KUKA KRL program: MyProgram_144().src

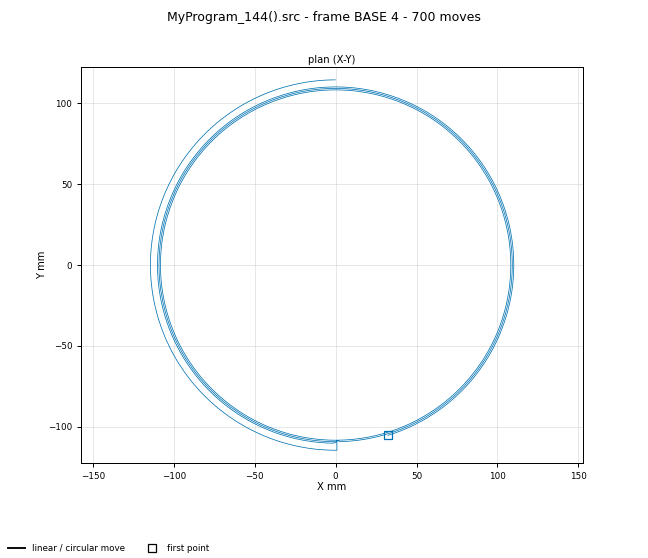
[picture p0: tool path of MyProgram_144().src in frame BASE 4, 700 of 700 moves have a stored position in this frame; points joined in program order, loops and branches not executed]
&ACCESS RVP
&REL 1
&PARAM TEMPLATE = C:\KRC\Roboter\Template\vorgabe
&PARAM EDITMASK = *
DEF MyProgram_144()
; ---- Setting reference (Base) ----
$BASE = BASE_DATA[4]

; --------------------------
; ---- Setting tool (TCP) ----
$TOOL = TOOL_DATA[3]
; --------------------------

$VEL.CP = VEL_APROX_PRINT
Startdeposition()
$VEL.CP = VEL_PRINT
LIN {X 32.3043,Y -105.2779,Z 114,A -76.1687,B 24.9494,C -1.6435,E1 25.049,E2 521.9318} C_DIS
LIN {X 36.8171,Y -103.7861,Z 114,A -73.6146,B 24.949,C -1.6502,E1 25.0557,E2 519.3669} C_DIS
LIN {X 40.1268,Y -102.5513,Z 114,A -71.7718,B 24.9488,C -1.6529,E1 25.0606,E2 517.5216} C_DIS
LIN {X 44.9405,Y -100.5354,Z 114,A -69.3366,B 24.9493,C -1.6447,E1 25.0667,E2 515.1116} C_DIS
LIN {X 48.2949,Y -98.9693,Z 114,A -67.5467,B 24.9495,C -1.6418,E1 25.0712,E2 513.3333} C_DIS
LIN {X 53.5849,Y -96.2059,Z 114,A -64.3362,B 24.9489,C -1.6518,E1 25.0792,E2 510.1083} C_DIS
LIN {X 56.8019,Y -94.3433,Z 114,A -62.2013,B 24.9481,C -1.6642,E1 25.0843,E2 507.9506} C_DIS
LIN {X 62.1001,Y -90.9432,Z 114,A -59.1184,B 24.9482,C -1.6622,E1 25.0915,E2 504.8827} C_DIS
LIN {X 65.0041,Y -88.8897,Z 114,A -57.5591,B 24.9488,C -1.6532,E1 25.095,E2 503.3502} C_DIS
LIN {X 67.0376,Y -87.3665,Z 114,A -55.8725,B 24.9476,C -1.6721,E1 25.0988,E2 501.6249} C_DIS
LIN {X 70.2691,Y -84.7891,Z 114,A -53.9266,B 24.9479,C -1.6678,E1 25.103,E2 499.6965} C_DIS
LIN {X 72.5045,Y -82.8856,Z 114,A -52.3507,B 24.9475,C -1.6735,E1 25.1063,E2 498.1135} C_DIS
LIN {X 75.3222,Y -80.3337,Z 114,A -50.387,B 24.9473,C -1.6775,E1 25.1104,E2 496.1481} C_DIS
LIN {X 77.8557,Y -77.8835,Z 114,A -48.461,B 24.9467,C -1.6861,E1 25.1142,E2 494.21} C_DIS
LIN {X 80.1666,Y -75.4999,Z 114,A -46.8371,B 24.9467,C -1.6859,E1 25.1174,E2 492.5937} C_DIS
LIN {X 82.7285,Y -72.6843,Z 114,A -44.8427,B 24.9464,C -1.6916,E1 25.1211,E2 490.5948} C_DIS
LIN {X 84.9909,Y -70.0262,Z 114,A -42.9743,B 24.9459,C -1.6987,E1 25.1244,E2 488.7181} C_DIS
LIN {X 87.034,Y -67.4692,Z 114,A -41.5863,B 24.9465,C -1.6892,E1 25.1268,E2 487.3591} C_DIS
LIN {X 88.7764,Y -65.1589,Z 114,A -39.9062,B 24.9458,C -1.7011,E1 25.1296,E2 485.6588} C_DIS
LIN {X 92.6081,Y -59.5874,Z 114,A -36.3603,B 24.9451,C -1.7122,E1 25.1352,E2 482.1042} C_DIS
LIN {X 95.3805,Y -55.0409,Z 114,A -33.6052,B 24.9446,C -1.7196,E1 25.1391,E2 479.346} C_DIS
LIN {X 97.1045,Y -51.9425,Z 114,A -30.8642,B 24.9416,C -1.7657,E1 25.1429,E2 476.5105} C_DIS
LIN {X 99.6138,Y -46.9497,Z 114,A -28.8531,B 24.9437,C -1.7337,E1 25.1452,E2 474.5857} C_DIS
LIN {X 100.9391,Y -44.025,Z 114,A -27.2776,B 24.9437,C -1.7345,E1 25.147,E2 473.0169} C_DIS
LIN {X 101.8876,Y -41.7839,Z 114,A -24.9103,B 24.94,C -1.7886,E1 25.1496,E2 470.535} C_DIS
LIN {X 104.1057,Y -35.9063,Z 114,A -21.5906,B 24.9392,C -1.8012,E1 25.1526,E2 467.2043} C_DIS
LIN {X 106.0459,Y -29.6867,Z 114,A -19.6143,B 24.9428,C -1.7475,E1 25.1541,E2 465.3661} C_DIS
LIN {X 106.6846,Y -27.3004,Z 114,A -17.8914,B 24.9412,C -1.7714,E1 25.1553,E2 463.5967} C_DIS
LIN {X 107.6606,Y -23.1559,Z 114,A -15.78,B 24.941,C -1.7738,E1 25.1566,E2 461.4918} C_DIS
LIN {X 108.3909,Y -19.4506,Z 114,A -13.9269,B 24.941,C -1.7751,E1 25.1575,E2 459.6465} C_DIS
LIN {X 109.0136,Y -15.5869,Z 114,A -11.905,B 24.9405,C -1.7811,E1 25.1584,E2 457.6225} C_DIS
LIN {X 109.4838,Y -11.8473,Z 114,A -10.1834,B 24.9408,C -1.7766,E1 25.1589,E2 455.9216} C_DIS
LIN {X 109.9148,Y -6.7857,Z 114,A -7.299,B 24.9395,C -1.7961,E1 25.1596,E2 453.0084} C_DIS
LIN {X 110.0683,Y -3.446,Z 114,A -5.6516,B 24.9395,C -1.7976,E1 25.1597,E2 451.3672} C_DIS
LIN {X 110.121,Y -0.6112,Z 114,A -3.8751,B 24.9382,C -1.816,E1 25.1597,E2 449.5578} C_DIS
LIN {X 110.0404,Y 4.2688,Z 114,A -1.5511,B 24.9382,C -1.8145,E1 25.1596,E2 447.2513} C_DIS
LIN {X 109.8312,Y 8.0234,Z 114,A 0.3876,B 24.9379,C -1.82,E1 25.1592,E2 445.3111} C_DIS
LIN {X 109.5211,Y 11.4902,Z 114,A 2.097,B 24.9379,C -1.8212,E1 25.1588,E2 443.609} C_DIS
LIN {X 109.109,Y 14.9152,Z 114,A 3.9492,B 24.9373,C -1.8295,E1 25.1581,E2 441.7481} C_DIS
LIN {X 108.6109,Y 18.1818,Z 114,A 5.5623,B 24.9373,C -1.8302,E1 25.1574,E2 440.1428} C_DIS
LIN {X 107.9638,Y 21.7008,Z 114,A 7.4442,B 24.9367,C -1.837,E1 25.1564,E2 438.256} C_DIS
LIN {X 107.3434,Y 24.5836,Z 114,A 8.962,B 24.9365,C -1.841,E1 25.1555,E2 436.7374} C_DIS
LIN {X 106.5404,Y 27.8614,Z 114,A 10.7334,B 24.936,C -1.8472,E1 25.1543,E2 434.9618} C_DIS
LIN {X 105.0229,Y 33.1235,Z 114,A 13.6108,B 24.9354,C -1.8571,E1 25.152,E2 432.0773} C_DIS
LIN {X 103.6854,Y 37.1036,Z 114,A 16.6543,B 24.9321,C -1.9024,E1 25.1491,E2 428.944} C_DIS
LIN {X 101.6602,Y 42.3358,Z 114,A 18.6311,B 24.9346,C -1.8684,E1 25.1471,E2 427.0584} C_DIS
LIN {X 100.4069,Y 45.2256,Z 114,A 20.2122,B 24.9344,C -1.8706,E1 25.1453,E2 425.4807} C_DIS
LIN {X 98.8908,Y 48.4539,Z 114,A 22.1571,B 24.9338,C -1.8798,E1 25.1429,E2 423.5245} C_DIS
LIN {X 97.2638,Y 51.6409,Z 114,A 24.2545,B 24.9326,C -1.8956,E1 25.1402,E2 421.4011} C_DIS
LIN {X 94.8756,Y 55.9067,Z 114,A 26.7935,B 24.9322,C -1.9022,E1 25.1366,E2 418.8594} C_DIS
LIN {X 92.3089,Y 60.0535,Z 114,A 29.0703,B 24.9325,C -1.8972,E1 25.1332,E2 416.6059} C_DIS
LIN {X 90.3472,Y 62.9628,Z 114,A 30.8213,B 24.9325,C -1.8986,E1 25.1305,E2 414.8602} C_DIS
LIN {X 88.2337,Y 65.8925,Z 114,A 32.6014,B 24.9325,C -1.8989,E1 25.1275,E2 413.088} C_DIS
LIN {X 84.6968,Y 70.3801,Z 114,A 35.6267,B 24.9317,C -1.9084,E1 25.1223,E2 410.0545} C_DIS
LIN {X 82.2831,Y 73.1882,Z 114,A 37.3292,B 24.9321,C -1.903,E1 25.1192,E2 408.3725} C_DIS
LIN {X 79.3562,Y 76.3512,Z 114,A 39.7796,B 24.9311,C -1.9171,E1 25.1145,E2 405.8994} C_DIS
LIN {X 76.8675,Y 78.8585,Z 114,A 41.7078,B 24.9305,C -1.9249,E1 25.1106,E2 403.9607} C_DIS
LIN {X 74.8797,Y 80.7482,Z 114,A 43.1989,B 24.9301,C -1.9307,E1 25.1075,E2 402.4622} C_DIS
LIN {X 71.615,Y 83.6557,Z 114,A 45.2986,B 24.9303,C -1.9276,E1 25.1032,E2 400.3781} C_DIS
LIN {X 68.7412,Y 86.0343,Z 114,A 47.3063,B 24.9299,C -1.9341,E1 25.0988,E2 398.3626} C_DIS
LIN {X 66.4134,Y 87.8424,Z 114,A 48.832,B 24.9297,C -1.9366,E1 25.0954,E2 396.8366} C_DIS
LIN {X 63.3023,Y 90.1112,Z 114,A 50.6227,B 24.9301,C -1.9308,E1 25.0914,E2 395.0658} C_DIS
LIN {X 60.4276,Y 92.0623,Z 114,A 52.8741,B 24.9285,C -1.953,E1 25.086,E2 392.7694} C_DIS
LIN {X 56.179,Y 94.7146,Z 114,A 55.3278,B 24.9287,C -1.9503,E1 25.0802,E2 390.3297} C_DIS
LIN {X 52.9765,Y 96.5437,Z 114,A 57.2821,B 24.9284,C -1.9545,E1 25.0754,E2 388.3712} C_DIS
LIN {X 48.8543,Y 98.6923,Z 114,A 59.4524,B 24.9289,C -1.947,E1 25.0701,E2 386.2246} C_DIS
LIN {X 45.5284,Y 100.2705,Z 114,A 61.4282,B 24.9286,C -1.9519,E1 25.0651,E2 384.2423} C_DIS
LIN {X 42.1119,Y 101.7542,Z 114,A 63.4155,B 24.9283,C -1.9561,E1 25.06,E2 382.2499} C_DIS
LIN {X 38.4349,Y 103.199,Z 114,A 66.0417,B 24.9263,C -1.9824,E1 25.053,E2 379.5669} C_DIS
LIN {X 34.2599,Y 104.6581,Z 114,A 67.6987,B 24.9282,C -1.9569,E1 25.0487,E2 377.9735} C_DIS
LIN {X 31.3328,Y 105.5707,Z 114,A 69.6145,B 24.9271,C -1.9717,E1 25.0435,E2 376.026} C_DIS
LIN {X 28.2462,Y 106.4392,Z 114,A 70.9701,B 24.928,C -1.9595,E1 25.0399,E2 374.7014} C_DIS
LIN {X 24.1237,Y 107.4495,Z 114,A 73.2559,B 24.9277,C -1.964,E1 25.0337,E2 372.4083} C_DIS
LIN {X 20.8233,Y 108.1356,Z 114,A 74.9128,B 24.9279,C -1.9607,E1 25.0292,E2 370.7611} C_DIS
LIN {X 16.9636,Y 108.8079,Z 114,A 76.9465,B 24.9279,C -1.9612,E1 25.0236,E2 368.7283} C_DIS
LIN {X 13.3331,Y 109.3134,Z 114,A 78.8773,B 24.9278,C -1.9626,E1 25.0182,E2 366.7957} C_DIS
LIN {X 9.9751,Y 109.6696,Z 114,A 80.606,B 24.9278,C -1.9617,E1 25.0134,E2 365.0704} C_DIS
LIN {X 6.296,Y 109.9423,Z 114,A 82.488,B 24.928,C -1.9601,E1 25.0082,E2 363.1928} C_DIS
LIN {X 2.8665,Y 110.0861,Z 114,A 84.3979,B 24.9276,C -1.9651,E1 25.0029,E2 361.2716} C_DIS
LIN {X -1.2189,Y 110.1168,Z 114,A 86.6393,B 24.9273,C -1.9694,E1 24.9966,E2 359.0199} C_DIS
LIN {X -5.4605,Y 109.9885,Z 114,A 88.6972,B 24.9278,C -1.9625,E1 24.9909,E2 356.978} C_DIS
LIN {X -8.5049,Y 109.7936,Z 114,A 90.2731,B 24.9278,C -1.9614,E1 24.9865,E2 355.4041} C_DIS
LIN {X -12.1976,Y 109.4464,Z 114,A 92.2543,B 24.9278,C -1.9625,E1 24.981,E2 353.4193} C_DIS
LIN {X -15.6118,Y 109.0101,Z 114,A 93.9501,B 24.9282,C -1.9575,E1 24.9763,E2 351.734} C_DIS
LIN {X -19.42,Y 108.3964,Z 114,A 95.7853,B 24.9288,C -1.9491,E1 24.9713,E2 349.9171} C_DIS
LIN {X -21.8574,Y 107.9317,Z 114,A 97.339,B 24.9281,C -1.9586,E1 24.967,E2 348.3389} C_DIS
LIN {X -26.1701,Y 106.9675,Z 114,A 100.5463,B 24.9255,C -1.9934,E1 24.9581,E2 345.0444} C_DIS
LIN {X -31.8564,Y 105.4153,Z 114,A 102.4384,B 24.9293,C -1.9424,E1 24.9533,E2 343.2705} C_DIS
LIN {X -37.6236,Y 103.4958,Z 114,A 105.8017,B 24.929,C -1.9465,E1 24.9444,E2 339.8911} C_DIS
LIN {X -40.94,Y 102.2311,Z 114,A 107.8444,B 24.9286,C -1.9518,E1 24.939,E2 337.8314} C_DIS
LIN {X -45.7047,Y 100.1911,Z 114,A 110.3935,B 24.9293,C -1.9419,E1 24.9325,E2 335.2997} C_DIS
LIN {X -48.9868,Y 98.6266,Z 114,A 112.713,B 24.9283,C -1.9559,E1 24.9266,E2 332.9408} C_DIS
LIN {X -52.1981,Y 96.9659,Z 114,A 114.2258,B 24.9296,C -1.9381,E1 24.923,E2 331.4662} C_DIS
LIN {X -55.7337,Y 94.9778,Z 114,A 116.2797,B 24.93,C -1.9321,E1 24.918,E2 329.4206} C_DIS
LIN {X -58.5565,Y 93.2637,Z 114,A 118.0509,B 24.93,C -1.931,E1 24.9138,E2 327.6464} C_DIS
LIN {X -61.885,Y 91.0888,Z 114,A 120.5693,B 24.9291,C -1.9446,E1 24.9079,E2 325.0872} C_DIS
LIN {X -64.9693,Y 88.9152,Z 114,A 122.0298,B 24.9308,C -1.9208,E1 24.9047,E2 323.6783} C_DIS
LIN {X -67.8244,Y 86.7588,Z 114,A 124.2205,B 24.9302,C -1.9297,E1 24.8998,E2 321.4584} C_DIS
LIN {X -71.8749,Y 83.4329,Z 114,A 127.1043,B 24.9302,C -1.9297,E1 24.8936,E2 318.5633} C_DIS
LIN {X -74.7712,Y 80.8477,Z 114,A 129.0145,B 24.9308,C -1.9207,E1 24.8897,E2 316.6669} C_DIS
LIN {X -78.7649,Y 76.9634,Z 114,A 131.8119,B 24.9316,C -1.9097,E1 24.8842,E2 313.8839} C_DIS
LIN {X -82.4622,Y 72.9882,Z 114,A 134.3424,B 24.933,C -1.8911,E1 24.8795,E2 311.3865} C_DIS
LIN {X -86.3423,Y 68.3515,Z 114,A 137.5194,B 24.9335,C -1.8841,E1 24.8739,E2 308.2116} C_DIS
LIN {X -89.6491,Y 63.9527,Z 114,A 140.4476,B 24.9338,C -1.8787,E1 24.869,E2 305.282} C_DIS
LIN {X -91.6855,Y 60.9991,Z 114,A 142.1773,B 24.9346,C -1.8683,E1 24.8663,E2 303.5687} C_DIS
LIN {X -94.787,Y 56.0565,Z 114,A 145.3711,B 24.9348,C -1.8656,E1 24.8616,E2 300.365} C_DIS
LIN {X -96.5285,Y 53.0045,Z 114,A 147.3129,B 24.9348,C -1.8646,E1 24.859,E2 298.4155} C_DIS
LIN {X -98.0542,Y 50.1226,Z 114,A 148.976,B 24.9353,C -1.8583,E1 24.8568,E2 296.7584} C_DIS
LIN {X -99.6777,Y 46.8124,Z 114,A 150.7436,B 24.9361,C -1.8467,E1 24.8547,E2 295.0088} C_DIS
LIN {X -101.664,Y 42.325,Z 114,A 153.4901,B 24.9361,C -1.8463,E1 24.8516,E2 292.2482} C_DIS
LIN {X -103.2769,Y 38.2238,Z 114,A 155.8023,B 24.9365,C -1.8399,E1 24.8493,E2 289.9382} C_DIS
LIN {X -104.3896,Y 35.0675,Z 114,A 157.4971,B 24.937,C -1.8327,E1 24.8478,E2 288.251} C_DIS
LIN {X -105.7838,Y 30.6115,Z 114,A 159.8834,B 24.9377,C -1.8233,E1 24.8459,E2 285.8732} C_DIS
LIN {X -107.2194,Y 25.1202,Z 114,A 162.9721,B 24.938,C -1.8191,E1 24.8437,E2 282.7767} C_DIS
LIN {X -107.9408,Y 21.8131,Z 114,A 164.6153,B 24.9387,C -1.8089,E1 24.8428,E2 281.148} C_DIS
LIN {X -108.5292,Y 18.6704,Z 114,A 166.8727,B 24.9375,C -1.8263,E1 24.8417,E2 278.8358} C_DIS
LIN {X -109.0902,Y 15.0478,Z 114,A 168.3564,B 24.939,C -1.8038,E1 24.8411,E2 277.3968} C_DIS
LIN {X -109.5684,Y 11.0388,Z 114,A 171.0753,B 24.9379,C -1.8208,E1 24.8403,E2 274.6212} C_DIS
LIN {X -109.9232,Y 6.6412,Z 114,A 172.611,B 24.9403,C -1.7842,E1 24.84,E2 273.1636} C_DIS
LIN {X -110.1166,Y 1.2654,Z 114,A 175.6442,B 24.9403,C -1.784,E1 24.8398,E2 270.1125} C_DIS
LIN {X -110.1145,Y -1.4343,Z 114,A 177.5079,B 24.9395,C -1.797,E1 24.8398,E2 268.2065} C_DIS
LIN {X -109.9939,Y -5.3508,Z 114,A 179.6017,B 24.9398,C -1.7926,E1 24.8402,E2 266.1107} C_DIS
LIN {X -109.7194,Y -9.4331,Z 114,A -178.7292,B 24.9414,C -1.768,E1 24.8405,E2 264.4901} C_DIS
LIN {X -109.4356,Y -12.2892,Z 114,A -176.8146,B 24.9407,C -1.7795,E1 24.8411,E2 262.5368} C_DIS
LIN {X -108.9413,Y -16.0959,Z 114,A -174.526,B 24.9403,C -1.7844,E1 24.8421,E2 260.2228} C_DIS
LIN {X -108.1152,Y -20.9288,Z 114,A -172.7875,B 24.9429,C -1.745,E1 24.8429,E2 258.5679} C_DIS
LIN {X -107.4211,Y -24.2447,Z 114,A -170.4746,B 24.9419,C -1.7607,E1 24.8444,E2 256.204} C_DIS
LIN {X -106.5292,Y -27.9049,Z 114,A -169.0976,B 24.9438,C -1.7322,E1 24.8453,E2 254.887} C_DIS
LIN {X -105.353,Y -32.0623,Z 114,A -166.6816,B 24.9438,C -1.7318,E1 24.8472,E2 252.458} C_DIS
LIN {X -104.4295,Y -34.9492,Z 114,A -165.129,B 24.9442,C -1.7261,E1 24.8485,E2 250.9101} C_DIS
LIN {X -103.2142,Y -38.3948,Z 114,A -163.1248,B 24.9442,C -1.7244,E1 24.8505,E2 248.8986} C_DIS
LIN {X -101.9882,Y -41.5368,Z 114,A -161.506,B 24.9449,C -1.714,E1 24.8521,E2 247.2955} C_DIS
LIN {X -100.8823,Y -44.1553,Z 114,A -159.764,B 24.9446,C -1.7199,E1 24.8541,E2 245.5297} C_DIS
LIN {X -98.8822,Y -48.4712,Z 114,A -157.6551,B 24.9459,C -1.6987,E1 24.8566,E2 243.4599} C_DIS
LIN {X -96.0493,Y -53.8654,Z 114,A -154.3168,B 24.9461,C -1.6964,E1 24.861,E2 240.1093} C_DIS
LIN {X -94.2141,Y -57.0145,Z 114,A -152.4164,B 24.9464,C -1.6915,E1 24.8637,E2 238.2109} C_DIS
LIN {X -92.8152,Y -59.2648,Z 114,A -150.2729,B 24.9447,C -1.718,E1 24.867,E2 235.9935} C_DIS
LIN {X -90.1561,Y -63.2377,Z 114,A -148.6355,B 24.9472,C -1.6782,E1 24.8695,E2 234.4428} C_DIS
LIN {X -86.1979,Y -68.5342,Z 114,A -144.9571,B 24.9472,C -1.679,E1 24.8757,E2 230.7448} C_DIS
LIN {X -83.7989,Y -71.4469,Z 114,A -143.0621,B 24.9476,C -1.6717,E1 24.8791,E2 228.8584} C_DIS
LIN {X -81.2882,Y -74.2912,Z 114,A -141.0843,B 24.9479,C -1.6674,E1 24.8828,E2 226.8821} C_DIS
LIN {X -78.8459,Y -76.8806,Z 114,A -139.1261,B 24.9479,C -1.6676,E1 24.8866,E2 224.9151} C_DIS
LIN {X -76.2978,Y -79.4077,Z 114,A -137.3686,B 24.9484,C -1.6593,E1 24.8901,E2 223.1699} C_DIS
LIN {X -73.573,Y -81.9387,Z 114,A -135.4544,B 24.9487,C -1.6546,E1 24.894,E2 221.2592} C_DIS
LIN {X -71.2807,Y -83.9404,Z 114,A -133.8601,B 24.9489,C -1.6519,E1 24.8974,E2 219.665} C_DIS
LIN {X -68.24,Y -86.4304,Z 114,A -131.7141,B 24.9489,C -1.6522,E1 24.9021,E2 217.5105} C_DIS
LIN {X -64.5235,Y -89.2394,Z 114,A -128.7329,B 24.9477,C -1.6704,E1 24.9089,E2 214.4754} C_DIS
LIN {X -61.0407,Y -91.658,Z 114,A -127.0719,B 24.9493,C -1.6447,E1 24.9126,E2 212.8698} C_DIS
LIN {X -58.565,Y -93.2584,Z 114,A -125.4735,B 24.9493,C -1.645,E1 24.9164,E2 211.2657} C_DIS
LIN {X -54.9688,Y -95.422,Z 114,A -123.3359,B 24.9496,C -1.64,E1 24.9215,E2 209.1337} C_DIS
LIN {X -51.4578,Y -97.3603,Z 114,A -121.2817,B 24.9499,C -1.6358,E1 24.9266,E2 207.0834} C_DIS
LIN {X -48.1628,Y -99.0329,Z 114,A -119.3115,B 24.9499,C -1.6354,E1 24.9315,E2 205.1092} C_DIS
LIN {X -44.9881,Y -100.5139,Z 114,A -117.4397,B 24.9499,C -1.6354,E1 24.9363,E2 203.2328} C_DIS
LIN {X -41.4514,Y -102.023,Z 114,A -114.8671,B 24.9486,C -1.6568,E1 24.9431,E2 200.6034} C_DIS
LIN {X -37.1934,Y -103.6527,Z 114,A -113.0418,B 24.9501,C -1.6321,E1 24.9477,E2 198.8332} C_DIS
LIN {X -34.4931,Y -104.5826,Z 114,A -111.2971,B 24.9495,C -1.6416,E1 24.9524,E2 197.0627} C_DIS
LIN {X -29.5647,Y -106.0805,Z 114,A -108.913,B 24.9504,C -1.6275,E1 24.9587,E2 194.7082} C_DIS
LIN {X -25.9792,Y -107.014,Z 114,A -107.0587,B 24.9506,C -1.6234,E1 24.9637,E2 192.8611} C_DIS
LIN {X -22.304,Y -107.84,Z 114,A -105.1248,B 24.9507,C -1.6214,E1 24.969,E2 190.9295} C_DIS
LIN {X -19.2869,Y -108.4203,Z 114,A -103.4094,B 24.9505,C -1.6257,E1 24.9737,E2 189.2021} C_DIS
LIN {X -15.5621,Y -109.0171,Z 114,A -101.7026,B 24.9512,C -1.6145,E1 24.9784,E2 187.5204} C_DIS
LIN {X -12.9079,Y -109.3632,Z 114,A -100.0154,B 24.9504,C -1.6266,E1 24.9831,E2 185.8033} C_DIS
LIN {X -8.8652,Y -109.7648,Z 114,A -98.0132,B 24.9507,C -1.6218,E1 24.9887,E2 183.8116} C_DIS
LIN {X -5.174,Y -110.0015,Z 114,A -95.9134,B 24.9503,C -1.6292,E1 24.9946,E2 181.6934} C_DIS
LIN {X -1.4311,Y -110.1144,Z 114,A -93.8231,B 24.9499,C -1.6356,E1 25.0005,E2 179.588} C_DIS
LIN {X -1.4311,Y -110.1144,Z 114,A -93.8231,B 24.9499,C -1.6356,E1 25.0005,E2 179.588} C_DIS
Enddeposition()
LIN {X 0.7939,Y -109.1989,Z 114,A -93.7268,B 24.9516,C -1.6074,E1 25.0005,E2 179.5585} C_DIS
Startdeposition()
$VEL.CP = VEL_PRINT
LIN {X -2.3355,Y -109.1788,Z 114,A -95.4072,B 24.9517,C -1.6054,E1 24.9958,E2 181.2435} C_DIS
LIN {X -5.5453,Y -109.0635,Z 114,A -97.1733,B 24.9519,C -1.6019,E1 24.9909,E2 183.0183} C_DIS
LIN {X -8.9577,Y -108.8356,Z 114,A -99.0359,B 24.9521,C -1.5992,E1 24.9857,E2 184.8882} C_DIS
LIN {X -13.2398,Y -108.3991,Z 114,A -101.142,B 24.9517,C -1.6057,E1 24.9799,E2 186.9802} C_DIS
LIN {X -16.5899,Y -107.9358,Z 114,A -102.9711,B 24.9517,C -1.6039,E1 24.9748,E2 188.8151} C_DIS
LIN {X -19.8828,Y -107.3795,Z 114,A -104.7313,B 24.9517,C -1.6041,E1 24.97,E2 190.5765} C_DIS
LIN {X -23.1749,Y -106.716,Z 114,A -106.4887,B 24.9517,C -1.6051,E1 24.9652,E2 192.3337} C_DIS
LIN {X -26.8944,Y -105.8402,Z 114,A -108.9002,B 24.9526,C -1.5899,E1 24.9585,E2 194.7847} C_DIS
LIN {X -30.1456,Y -104.9607,Z 114,A -110.0448,B 24.9511,C -1.616,E1 24.9556,E2 195.869} C_DIS
LIN {X -32.8817,Y -104.1368,Z 114,A -111.6886,B 24.9514,C -1.6113,E1 24.9512,E2 197.5269} C_DIS
LIN {X -35.7855,Y -103.1742,Z 114,A -113.4553,B 24.9517,C -1.6061,E1 24.9465,E2 199.3091} C_DIS
LIN {X -39.9101,Y -101.6491,Z 114,A -115.7497,B 24.9515,C -1.6088,E1 24.9405,E2 201.602} C_DIS
LIN {X -43.5494,Y -100.144,Z 114,A -117.8093,B 24.9514,C -1.6112,E1 24.9352,E2 203.6606} C_DIS
LIN {X -46.9166,Y -98.6122,Z 114,A -119.7309,B 24.9512,C -1.6143,E1 24.9303,E2 205.5798} C_DIS
LIN {X -49.9986,Y -97.0856,Z 114,A -121.5805,B 24.9512,C -1.6148,E1 24.9257,E2 207.4332} C_DIS
LIN {X -53.3124,Y -95.3056,Z 114,A -123.4281,B 24.9507,C -1.6224,E1 24.9212,E2 209.2678} C_DIS
LIN {X -56.1484,Y -93.6652,Z 114,A -125.305,B 24.9509,C -1.6186,E1 24.9166,E2 211.1594} C_DIS
LIN {X -58.983,Y -91.9041,Z 114,A -126.9357,B 24.9505,C -1.6261,E1 24.9128,E2 212.7775} C_DIS
LIN {X -65.0029,Y -87.7517,Z 114,A -130.7119,B 24.9499,C -1.6348,E1 24.9042,E2 216.5458} C_DIS
LIN {X -69.3844,Y -84.3295,Z 114,A -133.6115,B 24.9495,C -1.6408,E1 24.8979,E2 219.4419} C_DIS
LIN {X -71.6363,Y -82.4237,Z 114,A -135.3245,B 24.9498,C -1.6374,E1 24.8942,E2 221.1697} C_DIS
LIN {X -74.2905,Y -80.0417,Z 114,A -137.2983,B 24.9498,C -1.6372,E1 24.8901,E2 223.1519} C_DIS
LIN {X -76.8751,Y -77.5604,Z 114,A -139.0531,B 24.9492,C -1.646,E1 24.8866,E2 224.8931} C_DIS
LIN {X -79.4418,Y -74.9292,Z 114,A -141.0039,B 24.949,C -1.6494,E1 24.8828,E2 226.8444} C_DIS
LIN {X -81.8339,Y -72.3116,Z 114,A -142.9819,B 24.949,C -1.649,E1 24.8791,E2 228.8319} C_DIS
LIN {X -84.098,Y -69.6629,Z 114,A -144.6807,B 24.9485,C -1.6583,E1 24.8761,E2 230.5165} C_DIS
LIN {X -86.9831,Y -66.0273,Z 114,A -147.0336,B 24.9479,C -1.6673,E1 24.8721,E2 232.8591} C_DIS
LIN {X -89.2747,Y -62.8953,Z 114,A -149.3147,B 24.9482,C -1.663,E1 24.8683,E2 235.1614} C_DIS
LIN {X -91.7931,Y -59.1559,Z 114,A -151.292,B 24.9469,C -1.6839,E1 24.8653,E2 237.0988} C_DIS
LIN {X -93.1935,Y -56.9244,Z 114,A -153.0288,B 24.9475,C -1.6741,E1 24.8627,E2 238.868} C_DIS
LIN {X -95.124,Y -53.6376,Z 114,A -155.7701,B 24.9489,C -1.6517,E1 24.8588,E2 241.6771} C_DIS
LIN {X -97.4136,Y -49.3568,Z 114,A -157.6623,B 24.9469,C -1.6832,E1 24.8565,E2 243.5041} C_DIS
LIN {X -99.8127,Y -44.3076,Z 114,A -160.4272,B 24.946,C -1.6979,E1 24.8533,E2 246.2491} C_DIS
LIN {X -101.053,Y -41.397,Z 114,A -162.2443,B 24.946,C -1.6968,E1 24.8513,E2 248.0788} C_DIS
LIN {X -102.5023,Y -37.6658,Z 114,A -164.3022,B 24.9455,C -1.7046,E1 24.8493,E2 250.1298} C_DIS
LIN {X -103.5947,Y -34.5491,Z 114,A -165.9887,B 24.9451,C -1.7115,E1 24.8477,E2 251.8093} C_DIS
LIN {X -104.586,Y -31.4209,Z 114,A -167.9284,B 24.9453,C -1.7086,E1 24.8461,E2 253.7672} C_DIS
LIN {X -105.7309,Y -27.3196,Z 114,A -170.7595,B 24.9463,C -1.6934,E1 24.8441,E2 256.6512} C_DIS
LIN {X -106.8306,Y -22.6492,Z 114,A -172.4671,B 24.9438,C -1.7312,E1 24.8431,E2 258.2786} C_DIS
LIN {X -107.9957,Y -16.2027,Z 114,A -176.7896,B 24.9452,C -1.7093,E1 24.8411,E2 262.679} C_DIS
LIN {X -108.6034,Y -11.4311,Z 114,A -178.4529,B 24.9427,C -1.7492,E1 24.8406,E2 264.2571} C_DIS
LIN {X -109.0767,Y -5.2925,Z 114,A 177.3881,B 24.9442,C -1.7253,E1 24.8398,E2 268.4982} C_DIS
LIN {X -109.2033,Y -0.3688,Z 114,A 175.7642,B 24.9413,C -1.7691,E1 24.8398,E2 270.0274} C_DIS
LIN {X -109.021,Y 6.3133,Z 114,A 172.5904,B 24.9398,C -1.7928,E1 24.8401,E2 273.1635} C_DIS
LIN {X -108.5345,Y 12.0838,Z 114,A 168.9171,B 24.9407,C -1.7789,E1 24.841,E2 276.8921} C_DIS
LIN {X -107.8767,Y 16.9724,Z 114,A 166.5736,B 24.9395,C -1.7964,E1 24.8418,E2 279.2079} C_DIS
LIN {X -107.4356,Y 19.571,Z 114,A 165.0284,B 24.9396,C -1.7948,E1 24.8426,E2 280.766} C_DIS
LIN {X -106.7681,Y 22.9357,Z 114,A 163.1412,B 24.9394,C -1.7974,E1 24.8437,E2 282.6584} C_DIS
LIN {X -105.9807,Y 26.3378,Z 114,A 161.1165,B 24.9395,C -1.7961,E1 24.845,E2 284.6979} C_DIS
LIN {X -104.8025,Y 30.6912,Z 114,A 158.7995,B 24.9389,C -1.8054,E1 24.8467,E2 287.0061} C_DIS
LIN {X -103.6048,Y 34.5189,Z 114,A 156.8268,B 24.9381,C -1.8169,E1 24.8484,E2 288.9626} C_DIS
LIN {X -102.3543,Y 38.0706,Z 114,A 154.7463,B 24.938,C -1.8192,E1 24.8504,E2 291.0496} C_DIS
LIN {X -99.9336,Y 44.0321,Z 114,A 151.4627,B 24.937,C -1.833,E1 24.8539,E2 294.3185} C_DIS
LIN {X -98.7765,Y 46.5709,Z 114,A 149.8437,B 24.9371,C -1.8316,E1 24.8558,E2 295.9496} C_DIS
LIN {X -96.9463,Y 50.2712,Z 114,A 147.7502,B 24.9365,C -1.8408,E1 24.8584,E2 298.0325} C_DIS
LIN {X -95.3639,Y 53.208,Z 114,A 146.0447,B 24.936,C -1.8476,E1 24.8607,E2 299.7307} C_DIS
LIN {X -93.8346,Y 55.8619,Z 114,A 144.1599,B 24.9364,C -1.8419,E1 24.8634,E2 301.6389} C_DIS
LIN {X -91.1604,Y 60.1261,Z 114,A 141.8193,B 24.9351,C -1.8606,E1 24.8669,E2 303.9467} C_DIS
LIN {X -89.5537,Y 62.4944,Z 114,A 140.2919,B 24.9349,C -1.8638,E1 24.8693,E2 305.4741} C_DIS
LIN {X -87.2555,Y 65.6647,Z 114,A 137.8125,B 24.9356,C -1.8535,E1 24.8735,E2 307.9899} C_DIS
LIN {X -85.2341,Y 68.2708,Z 114,A 136.4023,B 24.9344,C -1.8701,E1 24.8759,E2 309.3673} C_DIS
LIN {X -83.0963,Y 70.8545,Z 114,A 134.6625,B 24.9341,C -1.8754,E1 24.879,E2 311.1024} C_DIS
LIN {X -79.5252,Y 74.8405,Z 114,A 131.6781,B 24.9341,C -1.8759,E1 24.8847,E2 314.0988} C_DIS
LIN {X -76.4856,Y 77.9451,Z 114,A 129.4495,B 24.9335,C -1.8833,E1 24.889,E2 316.3191} C_DIS
LIN {X -73.7287,Y 80.5572,Z 114,A 127.1999,B 24.9339,C -1.8783,E1 24.8937,E2 318.5898} C_DIS
LIN {X -71.3317,Y 82.6889,Z 114,A 125.7606,B 24.9329,C -1.8913,E1 24.8967,E2 320.0038} C_DIS
LIN {X -69.1607,Y 84.5129,Z 114,A 124.3023,B 24.9326,C -1.8957,E1 24.8998,E2 321.4572} C_DIS
LIN {X -66.4499,Y 86.6593,Z 114,A 122.574,B 24.9321,C -1.9029,E1 24.9036,E2 323.1747} C_DIS
LIN {X -63.67,Y 88.722,Z 114,A 120.6066,B 24.9323,C -1.9009,E1 24.908,E2 325.1538} C_DIS
LIN {X -60.1459,Y 91.1473,Z 114,A 118.4832,B 24.9316,C -1.91,E1 24.9129,E2 327.2627} C_DIS
LIN {X -57.4223,Y 92.8886,Z 114,A 116.6208,B 24.9318,C -1.9068,E1 24.9174,E2 329.1386} C_DIS
LIN {X -53.7489,Y 95.0619,Z 114,A 114.4833,B 24.9313,C -1.9147,E1 24.9225,E2 331.2636} C_DIS
LIN {X -50.8815,Y 96.6253,Z 114,A 112.6524,B 24.9313,C -1.9132,E1 24.927,E2 333.1033} C_DIS
LIN {X -47.845,Y 98.1661,Z 114,A 110.9053,B 24.9311,C -1.9175,E1 24.9314,E2 334.8446} C_DIS
LIN {X -43.6211,Y 100.1128,Z 114,A 108.595,B 24.9304,C -1.9263,E1 24.9372,E2 337.1398} C_DIS
LIN {X -40.5663,Y 101.391,Z 114,A 106.7103,B 24.9307,C -1.923,E1 24.9421,E2 339.0366} C_DIS
LIN {X -37.0734,Y 102.7184,Z 114,A 104.3713,B 24.9315,C -1.9109,E1 24.9483,E2 341.4091} C_DIS
LIN {X -33.6852,Y 103.8782,Z 114,A 102.9608,B 24.9301,C -1.9313,E1 24.952,E2 342.7735} C_DIS
LIN {X -27.0296,Y 105.8054,Z 114,A 99.3477,B 24.9297,C -1.9361,E1 24.9617,E2 346.3811} C_DIS
LIN {X -24.858,Y 106.3368,Z 114,A 97.709,B 24.931,C -1.9189,E1 24.9662,E2 348.0628} C_DIS
LIN {X -21.4313,Y 107.0811,Z 114,A 96.3942,B 24.9294,C -1.941,E1 24.9697,E2 349.3265} C_DIS
LIN {X -18.7652,Y 107.5805,Z 114,A 94.7266,B 24.93,C -1.9325,E1 24.9743,E2 351.0162} C_DIS
LIN {X -15.2243,Y 108.137,Z 114,A 92.9901,B 24.9295,C -1.9395,E1 24.9791,E2 352.7376} C_DIS
LIN {X -11.4957,Y 108.5966,Z 114,A 90.9998,B 24.9295,C -1.9398,E1 24.9846,E2 354.7284} C_DIS
LIN {X -8.1063,Y 108.9037,Z 114,A 89.2114,B 24.9295,C -1.9405,E1 24.9896,E2 356.5159} C_DIS
LIN {X -4.8187,Y 109.097,Z 114,A 87.423,B 24.9295,C -1.9387,E1 24.9946,E2 358.309} C_DIS
LIN {X -0.5292,Y 109.2021,Z 114,A 85.191,B 24.9295,C -1.9401,E1 25.0008,E2 360.5379} C_DIS
LIN {X 3.3908,Y 109.1507,Z 114,A 83.117,B 24.9295,C -1.9396,E1 25.0066,E2 362.6126} C_DIS
LIN {X 7.1519,Y 108.9691,Z 114,A 81.1518,B 24.9295,C -1.9401,E1 25.0121,E2 364.576} C_DIS
LIN {X 11.1621,Y 108.6315,Z 114,A 79.0971,B 24.9293,C -1.9422,E1 25.0178,E2 366.6246} C_DIS
LIN {X 14.6627,Y 108.2163,Z 114,A 77.0933,B 24.9298,C -1.9355,E1 25.0234,E2 368.6426} C_DIS
LIN {X 18.3913,Y 107.6442,Z 114,A 75.1648,B 24.9297,C -1.9369,E1 25.0287,E2 370.5658} C_DIS
LIN {X 22.0265,Y 106.9589,Z 114,A 73.3159,B 24.9295,C -1.9398,E1 25.0337,E2 372.4056} C_DIS
LIN {X 27.2046,Y 105.7604,Z 114,A 70.9539,B 24.9283,C -1.9558,E1 25.04,E2 374.7264} C_DIS
LIN {X 29.7728,Y 105.0664,Z 114,A 69.2404,B 24.9293,C -1.9417,E1 25.0447,E2 376.4704} C_DIS
LIN {X 32.6979,Y 104.1938,Z 114,A 67.5599,B 24.9296,C -1.9373,E1 25.0492,E2 378.1585} C_DIS
LIN {X 36.8526,Y 102.7989,Z 114,A 65.3672,B 24.9295,C -1.9397,E1 25.055,E2 380.3412} C_DIS
LIN {X 40.3013,Y 101.4955,Z 114,A 63.306,B 24.93,C -1.9325,E1 25.0604,E2 382.4148} C_DIS
LIN {X 43.6056,Y 100.1195,Z 114,A 61.3974,B 24.9302,C -1.9292,E1 25.0653,E2 384.3268} C_DIS
LIN {X 47.0707,Y 98.5382,Z 114,A 59.4572,B 24.9302,C -1.9292,E1 25.0702,E2 386.2619} C_DIS
LIN {X 50.1455,Y 97.0105,Z 114,A 57.563,B 24.9307,C -1.9231,E1 25.0749,E2 388.1656} C_DIS
LIN {X 53.3618,Y 95.278,Z 114,A 55.7563,B 24.9305,C -1.925,E1 25.0793,E2 389.9624} C_DIS
LIN {X 55.8393,Y 93.8479,Z 114,A 54.2266,B 24.9308,C -1.9216,E1 25.083,E2 391.4955} C_DIS
LIN {X 62.1303,Y 89.8067,Z 114,A 50.2671,B 24.9313,C -1.9137,E1 25.0923,E2 395.4605} C_DIS
LIN {X 65.6132,Y 87.2942,Z 114,A 48.1323,B 24.9313,C -1.9148,E1 25.0971,E2 397.5853} C_DIS
LIN {X 68.3355,Y 85.1817,Z 114,A 46.1987,B 24.9319,C -1.9061,E1 25.1013,E2 399.5322} C_DIS
LIN {X 71.0884,Y 82.8971,Z 114,A 44.3761,B 24.9319,C -1.9048,E1 25.1052,E2 401.3509} C_DIS
LIN {X 73.9008,Y 80.3993,Z 114,A 42.4979,B 24.9319,C -1.9048,E1 25.1091,E2 403.2214} C_DIS
LIN {X 76.5587,Y 77.873,Z 114,A 40.5112,B 24.9325,C -1.8981,E1 25.1131,E2 405.2158} C_DIS
LIN {X 79.0988,Y 75.2939,Z 114,A 38.4579,B 24.9332,C -1.8873,E1 25.1171,E2 407.2857} C_DIS
LIN {X 81.4426,Y 72.7494,Z 114,A 36.9028,B 24.9327,C -1.8944,E1 25.12,E2 408.8172} C_DIS
LIN {X 83.7942,Y 70.0284,Z 114,A 34.0209,B 24.936,C -1.8475,E1 25.1254,E2 411.7967} C_DIS
LIN {X 87.3121,Y 65.5893,Z 114,A 32.4172,B 24.9324,C -1.8989,E1 25.1279,E2 413.2714} C_DIS
LIN {X 88.7358,Y 63.6506,Z 114,A 30.7827,B 24.9338,C -1.8796,E1 25.1306,E2 414.9436} C_DIS
LIN {X 90.5519,Y 61.0391,Z 114,A 29.141,B 24.934,C -1.8765,E1 25.1332,E2 416.5846} C_DIS
LIN {X 92.4526,Y 58.1203,Z 114,A 27.2001,B 24.9347,C -1.8667,E1 25.1361,E2 418.5387} C_DIS
LIN {X 93.9719,Y 55.6295,Z 114,A 25.7704,B 24.9347,C -1.867,E1 25.1382,E2 419.9603} C_DIS
LIN {X 95.6416,Y 52.7107,Z 114,A 23.921,B 24.9353,C -1.8585,E1 25.1407,E2 421.8202} C_DIS
LIN {X 97.0975,Y 49.9753,Z 114,A 22.382,B 24.9353,C -1.8578,E1 25.1427,E2 423.3528} C_DIS
LIN {X 98.6447,Y 46.849,Z 114,A 20.5935,B 24.9355,C -1.8544,E1 25.1449,E2 425.1397} C_DIS
LIN {X 100.0497,Y 43.7657,Z 114,A 18.7579,B 24.9361,C -1.8468,E1 25.147,E2 426.9833} C_DIS
LIN {X 102.0354,Y 38.9128,Z 114,A 16.3521,B 24.9356,C -1.8538,E1 25.1495,E2 429.3592} C_DIS
LIN {X 103.3422,Y 35.298,Z 114,A 14.0272,B 24.9369,C -1.8342,E1 25.1517,E2 431.7173} C_DIS
LIN {X 104.83,Y 30.5979,Z 114,A 11.5839,B 24.937,C -1.8327,E1 25.1537,E2 434.1503} C_DIS
LIN {X 105.599,Y 27.8327,Z 114,A 10.0845,B 24.9373,C -1.8283,E1 25.1548,E2 435.6514} C_DIS
LIN {X 106.2456,Y 25.252,Z 114,A 8.5889,B 24.9379,C -1.8196,E1 25.1558,E2 437.1589} C_DIS
LIN {X 106.9612,Y 22.0152,Z 114,A 6.8928,B 24.9382,C -1.8161,E1 25.1567,E2 438.8535} C_DIS
LIN {X 107.6678,Y 18.2503,Z 114,A 4.8659,B 24.9387,C -1.809,E1 25.1578,E2 440.8852} C_DIS
LIN {X 108.2243,Y 14.6009,Z 114,A 2.8732,B 24.9393,C -1.8003,E1 25.1585,E2 442.8866} C_DIS
LIN {X 108.6422,Y 11.06,Z 114,A 1.0981,B 24.9393,C -1.7986,E1 25.1591,E2 444.6553} C_DIS
LIN {X 108.9408,Y 7.5702,Z 114,A -0.7212,B 24.9397,C -1.7935,E1 25.1595,E2 446.4759} C_DIS
LIN {X 109.1339,Y 3.9356,Z 114,A -2.685,B 24.9403,C -1.7849,E1 25.1597,E2 448.4483} C_DIS
LIN {X 109.2034,Y 0.3496,Z 114,A -4.3368,B 24.94,C -1.7889,E1 25.1597,E2 450.0806} C_DIS
LIN {X 109.1788,Y -2.3372,Z 114,A -5.8236,B 24.9406,C -1.781,E1 25.1597,E2 451.5774} C_DIS
LIN {X 109.0345,Y -6.0696,Z 114,A -7.8062,B 24.941,C -1.7736,E1 25.1595,E2 453.5656} C_DIS
LIN {X 108.7316,Y -10.1399,Z 114,A -9.8115,B 24.9411,C -1.7726,E1 25.159,E2 455.5612} C_DIS
LIN {X 108.4063,Y -13.1781,Z 114,A -11.6464,B 24.9421,C -1.7571,E1 25.1584,E2 457.4218} C_DIS
LIN {X 107.8813,Y -16.9425,Z 114,A -13.6155,B 24.9425,C -1.7518,E1 25.1576,E2 459.3919} C_DIS
LIN {X 107.225,Y -20.6922,Z 114,A -15.4931,B 24.9425,C -1.7506,E1 25.1567,E2 461.2613} C_DIS
LIN {X 106.4494,Y -24.3706,Z 114,A -18.1503,B 24.9449,C -1.7142,E1 25.155,E2 463.989} C_DIS
LIN {X 105.3356,Y -28.8079,Z 114,A -19.5445,B 24.9426,C -1.7508,E1 25.1541,E2 465.2888} C_DIS
LIN {X 104.5471,Y -31.5518,Z 114,A -21.34,B 24.9437,C -1.7328,E1 25.1527,E2 467.1164} C_DIS
LIN {X 103.7598,Y -34.0509,Z 114,A -22.7822,B 24.9442,C -1.7255,E1 25.1514,E2 468.5678} C_DIS
LIN {X 102.5837,Y -37.4426,Z 114,A -24.981,B 24.9455,C -1.7058,E1 25.1493,E2 470.8008} C_DIS
LIN {X 101.3427,Y -40.6854,Z 114,A -26.2332,B 24.9442,C -1.7252,E1 25.1481,E2 472.0003} C_DIS
LIN {X 100.0959,Y -43.6597,Z 114,A -28.0468,B 24.9449,C -1.7146,E1 25.1461,E2 473.8289} C_DIS
LIN {X 98.752,Y -46.6237,Z 114,A -30.0586,B 24.9461,C -1.696,E1 25.1437,E2 475.8737} C_DIS
LIN {X 96.5076,Y -51.1048,Z 114,A -32.2943,B 24.9455,C -1.7055,E1 25.1409,E2 478.0752} C_DIS
LIN {X 95.2023,Y -53.4974,Z 114,A -33.7969,B 24.946,C -1.698,E1 25.1388,E2 479.5875} C_DIS
LIN {X 92.6348,Y -57.8287,Z 114,A -36.9359,B 24.9478,C -1.6687,E1 25.1342,E2 482.7798} C_DIS
LIN {X 90.534,Y -61.0655,Z 114,A -38.71,B 24.9475,C -1.6739,E1 25.1314,E2 484.5328} C_DIS
LIN {X 88.4212,Y -64.0884,Z 114,A -40.6071,B 24.9477,C -1.6701,E1 25.1284,E2 486.4295} C_DIS
LIN {X 85.7995,Y -67.5562,Z 114,A -42.6219,B 24.9474,C -1.6756,E1 25.125,E2 488.4219} C_DIS
LIN {X 83.5651,Y -70.3041,Z 114,A -44.5746,B 24.948,C -1.6665,E1 25.1215,E2 490.387} C_DIS
LIN {X 81.2722,Y -72.9397,Z 114,A -46.3197,B 24.948,C -1.6656,E1 25.1182,E2 492.1263} C_DIS
LIN {X 78.6411,Y -75.769,Z 114,A -48.3242,B 24.9483,C -1.6615,E1 25.1144,E2 494.1318} C_DIS
LIN {X 75.9534,Y -78.4634,Z 114,A -50.2979,B 24.9485,C -1.6576,E1 25.1105,E2 496.1065} C_DIS
LIN {X 73.685,Y -80.5973,Z 114,A -51.9523,B 24.9488,C -1.6529,E1 25.1071,E2 497.7654} C_DIS
LIN {X 70.8299,Y -83.1173,Z 114,A -53.9298,B 24.949,C -1.6492,E1 25.1029,E2 499.7438} C_DIS
LIN {X 67.8496,Y -85.5677,Z 114,A -56.3602,B 24.9504,C -1.6272,E1 25.0975,E2 502.217} C_DIS
LIN {X 65.0156,Y -87.7417,Z 114,A -57.651,B 24.9491,C -1.6483,E1 25.0948,E2 503.4533} C_DIS
LIN {X 62.8357,Y -89.3164,Z 114,A -59.6774,B 24.9509,C -1.6189,E1 25.09,E2 505.5422} C_DIS
LIN {X 59.8312,Y -91.3549,Z 114,A -61.0749,B 24.9498,C -1.6369,E1 25.0868,E2 506.8924} C_DIS
LIN {X 56.7408,Y -93.3051,Z 114,A -62.9822,B 24.95,C -1.6336,E1 25.0823,E2 508.8013} C_DIS
LIN {X 53.5169,Y -95.1914,Z 114,A -64.9931,B 24.9503,C -1.6279,E1 25.0774,E2 510.8198} C_DIS
LIN {X 49.2734,Y -97.4562,Z 114,A -67.2022,B 24.9498,C -1.637,E1 25.072,E2 513.0011} C_DIS
LIN {X 45.9339,Y -99.073,Z 114,A -69.3509,B 24.9505,C -1.6253,E1 25.0666,E2 515.172} C_DIS
LIN {X 40.858,Y -101.2724,Z 114,A -72.1465,B 24.9505,C -1.6255,E1 25.0594,E2 517.9605} C_DIS
LIN {X 37.4595,Y -102.5775,Z 114,A -74.2146,B 24.9511,C -1.6161,E1 25.054,E2 520.0462} C_DIS
LIN {X 33.9084,Y -103.8059,Z 114,A -77.0943,B 24.9535,C -1.5756,E1 25.0461,E2 523.0163} C_DIS
LIN {X 28.6125,Y -105.3884,Z 114,A -79.0672,B 24.9514,C -1.6112,E1 25.041,E2 524.9018} C_DIS
LIN {X 25.3451,Y -106.2229,Z 114,A -80.8843,B 24.9516,C -1.6073,E1 25.0361,E2 526.7252} C_DIS
LIN {X 21.9681,Y -106.9709,Z 114,A -82.6113,B 24.9515,C -1.6094,E1 25.0314,E2 528.4451} C_DIS
LIN {X 18.388,Y -107.6448,Z 114,A -84.5911,B 24.9517,C -1.605,E1 25.0259,E2 530.4332} C_DIS
LIN {X 14.5708,Y -108.2282,Z 114,A -86.6275,B 24.9518,C -1.6031,E1 25.0203,E2 532.4722} C_DIS
LIN {X 10.7687,Y -108.6726,Z 114,A -88.6876,B 24.952,C -1.5998,E1 25.0145,E2 534.5388} C_DIS
LIN {X 6.8016,Y -108.9928,Z 114,A -90.7918,B 24.9521,C -1.5982,E1 25.0087,E2 536.6458} C_DIS
LIN {X 2.6759,Y -109.1726,Z 114,A -92.8329,B 24.9519,C -1.6026,E1 25.003,E2 538.6759} C_DIS
LIN {X 2.6759,Y -109.1726,Z 114,A -92.8329,B 24.9519,C -1.6026,E1 25.003,E2 538.6759} C_DIS
Enddeposition()
LIN {X 0.7824,Y -108.2811,Z 114,A -93.1785,B 24.9493,C -1.6453,E1 25.0023,E2 538.9204} C_DIS
Startdeposition()
$VEL.CP = VEL_PRINT
LIN {X 3.2968,Y -108.2342,Z 114,A -91.8053,B 24.9491,C -1.6474,E1 25.0062,E2 537.5423} C_DIS
LIN {X 5.9454,Y -108.1211,Z 114,A -90.3923,B 24.9491,C -1.6484,E1 25.0101,E2 536.1275} C_DIS
LIN {X 8.5901,Y -107.9431,Z 114,A -88.9913,B 24.9491,C -1.649,E1 25.014,E2 534.7258} C_DIS
LIN {X 11.2289,Y -107.7006,Z 114,A -87.5837,B 24.949,C -1.65,E1 25.0179,E2 533.3167} C_DIS
LIN {X 13.8913,Y -107.3897,Z 114,A -86.1854,B 24.949,C -1.65,E1 25.0218,E2 531.9193} C_DIS
LIN {X 16.5633,Y -107.0101,Z 114,A -84.7596,B 24.949,C -1.651,E1 25.0257,E2 530.4926} C_DIS
LIN {X 19.1793,Y -106.5723,Z 114,A -83.2768,B 24.9486,C -1.6554,E1 25.0299,E2 529.0009} C_DIS
LIN {X 22.8663,Y -105.8427,Z 114,A -81.3188,B 24.9486,C -1.6559,E1 25.0352,E2 527.0443} C_DIS
LIN {X 25.6884,Y -105.1932,Z 114,A -79.8443,B 24.9486,C -1.6549,E1 25.0392,E2 525.5742} C_DIS
LIN {X 28.2125,Y -104.5446,Z 114,A -78.444,B 24.9486,C -1.6573,E1 25.043,E2 524.1704} C_DIS
LIN {X 30.8106,Y -103.8086,Z 114,A -77.0348,B 24.9485,C -1.6581,E1 25.0468,E2 522.7617} C_DIS
LIN {X 33.3268,Y -103.0283,Z 114,A -75.6296,B 24.9483,C -1.6602,E1 25.0505,E2 521.3541} C_DIS
LIN {X 36.4694,Y -101.9604,Z 114,A -73.9007,B 24.9483,C -1.6613,E1 25.0551,E2 519.6261} C_DIS
LIN {X 38.9399,Y -101.0425,Z 114,A -72.5104,B 24.9482,C -1.663,E1 25.0587,E2 518.2347} C_DIS
LIN {X 41.9631,Y -99.8229,Z 114,A -70.7823,B 24.948,C -1.6657,E1 25.0632,E2 516.5043} C_DIS
LIN {X 44.9539,Y -98.5135,Z 114,A -69.0614,B 24.9479,C -1.668,E1 25.0676,E2 514.7821} C_DIS
LIN {X 47.491,Y -97.3167,Z 114,A -67.5897,B 24.9477,C -1.6699,E1 25.0713,E2 513.3099} C_DIS
LIN {X 50.3131,Y -95.886,Z 114,A -65.8815,B 24.9475,C -1.6742,E1 25.0755,E2 511.5962} C_DIS
LIN {X 52.8171,Y -94.5297,Z 114,A -64.3745,B 24.9473,C -1.6769,E1 25.0792,E2 510.0872} C_DIS
LIN {X 55.6616,Y -92.8855,Z 114,A -62.6888,B 24.9473,C -1.6778,E1 25.0833,E2 508.4046} C_DIS
LIN {X 57.9148,Y -91.4976,Z 114,A -61.2945,B 24.9471,C -1.6802,E1 25.0866,E2 507.009} C_DIS
LIN {X 60.1318,Y -90.0559,Z 114,A -59.901,B 24.9469,C -1.6827,E1 25.0898,E2 505.6141} C_DIS
LIN {X 62.8272,Y -88.1944,Z 114,A -58.177,B 24.9467,C -1.6859,E1 25.0938,E2 503.8885} C_DIS
LIN {X 65.5385,Y -86.2009,Z 114,A -56.1241,B 24.9457,C -1.7015,E1 25.0984,E2 501.8062} C_DIS
LIN {X 68.941,Y -83.5031,Z 114,A -54.017,B 24.9459,C -1.6983,E1 25.103,E2 499.7146} C_DIS
LIN {X 71.4841,Y -81.3366,Z 114,A -52.1999,B 24.9456,C -1.7045,E1 25.1068,E2 497.8899} C_DIS
LIN {X 74.1868,Y -78.8786,Z 114,A -50.369,B 24.9456,C -1.7047,E1 25.1105,E2 496.0661} C_DIS
LIN {X 76.7942,Y -76.3432,Z 114,A -48.4204,B 24.9452,C -1.7104,E1 25.1144,E2 494.1121} C_DIS
LIN {X 79.0959,Y -73.9558,Z 114,A -46.6114,B 24.9447,C -1.7172,E1 25.1179,E2 492.295} C_DIS
LIN {X 81.562,Y -71.226,Z 114,A -44.7772,B 24.9447,C -1.7173,E1 25.1213,E2 490.4688} C_DIS
LIN {X 83.923,Y -68.4291,Z 114,A -42.8213,B 24.9443,C -1.7233,E1 25.1248,E2 488.5078} C_DIS
LIN {X 85.965,Y -65.8455,Z 114,A -41.1224,B 24.9442,C -1.7261,E1 25.1277,E2 486.8103} C_DIS
LIN {X 87.9289,Y -63.1993,Z 114,A -39.3527,B 24.9438,C -1.732,E1 25.1306,E2 485.0351} C_DIS
LIN {X 89.6003,Y -60.8055,Z 114,A -37.7954,B 24.9435,C -1.7369,E1 25.1331,E2 483.4739} C_DIS
LIN {X 91.579,Y -57.7844,Z 114,A -36.0958,B 24.9437,C -1.733,E1 25.1356,E2 481.792} C_DIS
LIN {X 92.8847,Y -55.6629,Z 114,A -34.6185,B 24.943,C -1.7439,E1 25.1378,E2 480.2967} C_DIS
LIN {X 94.5298,Y -52.8169,Z 114,A -32.9635,B 24.943,C -1.7453,E1 25.1401,E2 478.647} C_DIS
LIN {X 95.7931,Y -50.4895,Z 114,A -31.5711,B 24.9427,C -1.749,E1 25.1419,E2 477.253} C_DIS
LIN {X 96.9987,Y -48.1327,Z 114,A -30.1794,B 24.9424,C -1.7528,E1 25.1437,E2 475.8597} C_DIS
LIN {X 98.2815,Y -45.4568,Z 114,A -28.5845,B 24.942,C -1.7587,E1 25.1456,E2 474.2597} C_DIS
LIN {X 99.527,Y -42.6652,Z 114,A -27.0225,B 24.9419,C -1.7612,E1 25.1473,E2 472.7004} C_DIS
LIN {X 100.5422,Y -40.2145,Z 114,A -25.6182,B 24.9416,C -1.7655,E1 25.1488,E2 471.2934} C_DIS
LIN {X 101.5058,Y -37.716,Z 114,A -24.2184,B 24.9413,C -1.7692,E1 25.1502,E2 469.8928} C_DIS
LIN {X 102.5162,Y -34.8715,Z 114,A -22.55,B 24.9408,C -1.7774,E1 25.1517,E2 468.2145} C_DIS
LIN {X 103.4143,Y -32.1092,Z 114,A -21.0984,B 24.9408,C -1.7785,E1 25.1529,E2 466.7686} C_DIS
LIN {X 104.1776,Y -29.5387,Z 114,A -19.6936,B 24.9405,C -1.7824,E1 25.154,E2 465.3627} C_DIS
LIN {X 104.8584,Y -27.0227,Z 114,A -18.3375,B 24.9402,C -1.7858,E1 25.155,E2 464.0064} C_DIS
LIN {X 105.4839,Y -24.4678,Z 114,A -16.8774,B 24.9397,C -1.7933,E1 25.1559,E2 462.5371} C_DIS
LIN {X 106.2083,Y -21.1124,Z 114,A -15.1441,B 24.9396,C -1.7954,E1 25.1569,E2 460.8088} C_DIS
LIN {X 106.6935,Y -18.5048,Z 114,A -13.7503,B 24.9393,C -1.7995,E1 25.1576,E2 459.4135} C_DIS
LIN {X 107.1148,Y -15.8858,Z 114,A -12.3565,B 24.939,C -1.8036,E1 25.1582,E2 458.0182} C_DIS
LIN {X 107.52,Y -12.8462,Z 114,A -10.6695,B 24.9385,C -1.8118,E1 25.1588,E2 456.3219} C_DIS
LIN {X 107.8234,Y -9.9812,Z 114,A -9.2151,B 24.9383,C -1.8136,E1 25.1592,E2 454.8717} C_DIS
LIN {X 108.0368,Y -7.318,Z 114,A -7.8163,B 24.9381,C -1.8176,E1 25.1595,E2 453.4719} C_DIS
LIN {X 108.1856,Y -4.6239,Z 114,A -6.4095,B 24.9378,C -1.8213,E1 25.1597,E2 452.0647} C_DIS
LIN {X 108.2656,Y -2.0197,Z 114,A -5.0948,B 24.9378,C -1.8229,E1 25.1597,E2 450.7539} C_DIS
LIN {X 108.2849,Y 0.2597,Z 114,A -3.9377,B 24.9376,C -1.8247,E1 25.1597,E2 449.5996} C_DIS
LIN {X 108.2357,Y 3.2479,Z 114,A -2.258,B 24.9369,C -1.8342,E1 25.1597,E2 447.9076} C_DIS
LIN {X 108.1204,Y 5.9579,Z 114,A -0.8358,B 24.9367,C -1.8382,E1 25.1595,E2 446.4842} C_DIS
LIN {X 107.942,Y 8.6049,Z 114,A 0.5583,B 24.9364,C -1.8423,E1 25.1592,E2 445.0887} C_DIS
LIN {X 107.6556,Y 11.6588,Z 114,A 2.2809,B 24.9357,C -1.8519,E1 25.1587,E2 443.3537} C_DIS
LIN {X 107.21,Y 15.2157,Z 114,A 4.0538,B 24.9357,C -1.8525,E1 25.1581,E2 441.5899} C_DIS
LIN {X 106.7975,Y 17.8828,Z 114,A 5.4612,B 24.9354,C -1.8561,E1 25.1574,E2 440.1822} C_DIS
LIN {X 106.3275,Y 20.4934,Z 114,A 6.9136,B 24.935,C -1.8627,E1 25.1567,E2 438.7227} C_DIS
LIN {X 105.5713,Y 24.0894,Z 114,A 8.8759,B 24.9345,C -1.8696,E1 25.1555,E2 436.7557} C_DIS
LIN {X 104.8694,Y 26.9798,Z 114,A 10.3438,B 24.9345,C -1.8698,E1 25.1545,E2 435.2958} C_DIS
LIN {X 104.1802,Y 29.5297,Z 114,A 11.719,B 24.9342,C -1.8731,E1 25.1535,E2 433.9207} C_DIS
LIN {X 103.4463,Y 32.0058,Z 114,A 13.1087,B 24.9339,C -1.8783,E1 25.1524,E2 432.5267} C_DIS
LIN {X 102.6162,Y 34.575,Z 114,A 14.5148,B 24.9336,C -1.8816,E1 25.1511,E2 431.1207} C_DIS
LIN {X 101.7243,Y 37.117,Z 114,A 15.9198,B 24.9334,C -1.8849,E1 25.1498,E2 429.7157} C_DIS
LIN {X 100.8037,Y 39.549,Z 114,A 17.317,B 24.933,C -1.8899,E1 25.1484,E2 428.3145} C_DIS
LIN {X 99.7926,Y 42.035,Z 114,A 18.7211,B 24.9328,C -1.8934,E1 25.1469,E2 426.9099} C_DIS
LIN {X 98.7331,Y 44.4667,Z 114,A 20.1161,B 24.9325,C -1.8971,E1 25.1453,E2 425.5139} C_DIS
LIN {X 97.6143,Y 46.8718,Z 114,A 21.511,B 24.9323,C -1.9007,E1 25.1436,E2 424.118} C_DIS
LIN {X 96.219,Y 49.6751,Z 114,A 23.1694,B 24.9319,C -1.9054,E1 25.1415,E2 422.4573} C_DIS
LIN {X 94.8618,Y 52.2223,Z 114,A 24.6632,B 24.9317,C -1.9081,E1 25.1396,E2 420.9649} C_DIS
LIN {X 93.3171,Y 54.9314,Z 114,A 26.3619,B 24.9313,C -1.9147,E1 25.1372,E2 419.2593} C_DIS
LIN {X 91.8178,Y 57.402,Z 114,A 27.8236,B 24.9312,C -1.9158,E1 25.135,E2 417.8024} C_DIS
LIN {X 90.4154,Y 59.5866,Z 114,A 29.203,B 24.9309,C -1.9197,E1 25.1329,E2 416.4208} C_DIS
LIN {X 88.9023,Y 61.8214,Z 114,A 30.6008,B 24.9307,C -1.922,E1 25.1307,E2 415.0244} C_DIS
LIN {X 87.2615,Y 64.1168,Z 114,A 32.1542,B 24.9303,C -1.9284,E1 25.1282,E2 413.4635} C_DIS
LIN {X 85.0349,Y 67.0417,Z 114,A 34.1308,B 24.9298,C -1.9345,E1 25.1248,E2 411.4818} C_DIS
LIN {X 82.6354,Y 69.9786,Z 114,A 36.1218,B 24.9295,C -1.9386,E1 25.1212,E2 409.4904} C_DIS
LIN {X 80.45,Y 72.4805,Z 114,A 37.9429,B 24.9291,C -1.9453,E1 25.1178,E2 407.6615} C_DIS
LIN {X 77.9615,Y 75.15,Z 114,A 39.7647,B 24.9291,C -1.9449,E1 25.1144,E2 405.8486} C_DIS
LIN {X 75.3955,Y 77.7248,Z 114,A 41.7138,B 24.9287,C -1.9501,E1 25.1105,E2 403.8954} C_DIS
LIN {X 72.9642,Y 80.0116,Z 114,A 43.5264,B 24.9283,C -1.9557,E1 25.1067,E2 402.0769} C_DIS
LIN {X 70.2251,Y 82.4254,Z 114,A 45.3634,B 24.9283,C -1.9555,E1 25.1029,E2 400.2477} C_DIS
LIN {X 67.4117,Y 84.7425,Z 114,A 47.3162,B 24.928,C -1.9601,E1 25.0986,E2 398.2912} C_DIS
LIN {X 65.0608,Y 86.5599,Z 114,A 48.8303,B 24.928,C -1.9605,E1 25.0953,E2 396.7818} C_DIS
LIN {X 62.391,Y 88.5057,Z 114,A 50.6989,B 24.9273,C -1.9686,E1 25.091,E2 394.9005} C_DIS
LIN {X 59.3247,Y 90.5881,Z 114,A 52.4515,B 24.9278,C -1.963,E1 25.087,E2 393.1671} C_DIS
LIN {X 56.5084,Y 92.371,Z 114,A 54.3219,B 24.9272,C -1.9702,E1 25.0825,E2 391.2855} C_DIS
LIN {X 53.6758,Y 94.0453,Z 114,A 56.0074,B 24.9272,C -1.9704,E1 25.0785,E2 389.6047} C_DIS
LIN {X 51.0541,Y 95.4956,Z 114,A 57.6459,B 24.9269,C -1.9748,E1 25.0744,E2 387.9605} C_DIS
LIN {X 48.1087,Y 97.0107,Z 114,A 59.3138,B 24.9269,C -1.9735,E1 25.0703,E2 386.3002} C_DIS
LIN {X 45.7108,Y 98.1633,Z 114,A 60.716,B 24.9269,C -1.975,E1 25.0668,E2 384.8981} C_DIS
LIN {X 43.2926,Y 99.2535,Z 114,A 62.1162,B 24.9268,C -1.9765,E1 25.0632,E2 383.4978} C_DIS
LIN {X 40.4221,Y 100.4577,Z 114,A 63.7652,B 24.9266,C -1.9782,E1 25.0589,E2 381.8485} C_DIS
LIN {X 37.7369,Y 101.4981,Z 114,A 65.2697,B 24.9266,C -1.9789,E1 25.055,E2 380.3457} C_DIS
LIN {X 34.9241,Y 102.4985,Z 114,A 66.9522,B 24.9262,C -1.9846,E1 25.0505,E2 378.6531} C_DIS
LIN {X 31.6755,Y 103.5487,Z 114,A 68.6686,B 24.9263,C -1.9823,E1 25.046,E2 376.9452} C_DIS
LIN {X 28.8972,Y 104.3594,Z 114,A 70.2767,B 24.926,C -1.9865,E1 25.0416,E2 375.3299} C_DIS
LIN {X 25.7204,Y 105.1854,Z 114,A 71.9178,B 24.9262,C -1.9836,E1 25.0372,E2 373.6981} C_DIS
LIN {X 22.6223,Y 105.896,Z 114,A 73.752,B 24.9257,C -1.9907,E1 25.0322,E2 371.8495} C_DIS
LIN {X 19.1853,Y 106.5712,Z 114,A 75.4441,B 24.9261,C -1.9849,E1 25.0276,E2 370.1731} C_DIS
LIN {X 16.5692,Y 107.0092,Z 114,A 76.8585,B 24.9261,C -1.9858,E1 25.0237,E2 368.758} C_DIS
LIN {X 13.8971,Y 107.3889,Z 114,A 78.3181,B 24.9259,C -1.9874,E1 25.0196,E2 367.2958} C_DIS
LIN {X 10.3682,Y 107.7877,Z 114,A 80.1643,B 24.926,C -1.9863,E1 25.0145,E2 365.4533} C_DIS
LIN {X 7.3238,Y 108.0364,Z 114,A 81.7803,B 24.926,C -1.9864,E1 25.01,E2 363.8379} C_DIS
LIN {X 4.629,Y 108.1854,Z 114,A 83.1974,B 24.926,C -1.9859,E1 25.0061,E2 362.4224} C_DIS
LIN {X 2.0241,Y 108.2655,Z 114,A 84.6475,B 24.9259,C -1.9886,E1 25.002,E2 360.9662} C_DIS
LIN {X -1.3269,Y 108.2783,Z 114,A 86.354,B 24.9261,C -1.9855,E1 24.9973,E2 359.2671} C_DIS
LIN {X -3.9886,Y 108.2129,Z 114,A 87.7599,B 24.9261,C -1.985,E1 24.9933,E2 357.8623} C_DIS
LIN {X -7.1342,Y 108.0493,Z 114,A 89.4675,B 24.9261,C -1.986,E1 24.9886,E2 356.1516} C_DIS
LIN {X -9.9665,Y 107.8248,Z 114,A 91.0063,B 24.926,C -1.9867,E1 24.9843,E2 354.6104} C_DIS
LIN {X -13.4528,Y 107.4465,Z 114,A 92.851,B 24.9261,C -1.9852,E1 24.9792,E2 352.7681} C_DIS
LIN {X -16.5684,Y 107.0093,Z 114,A 94.4584,B 24.9264,C -1.9819,E1 24.9747,E2 351.1674} C_DIS
LIN {X -19.1845,Y 106.5714,Z 114,A 95.8642,B 24.9264,C -1.9809,E1 24.9709,E2 349.7624} C_DIS
LIN {X -21.7435,Y 106.0789,Z 114,A 97.2567,B 24.9264,C -1.9803,E1 24.9671,E2 348.3697} C_DIS
LIN {X -24.3617,Y 105.5084,Z 114,A 98.6731,B 24.9266,C -1.979,E1 24.9632,E2 346.9547} C_DIS
LIN {X -26.9489,Y 104.8774,Z 114,A 100.0613,B 24.9267,C -1.9768,E1 24.9595,E2 345.5698} C_DIS
LIN {X -29.4662,Y 104.1981,Z 114,A 101.5692,B 24.9265,C -1.9804,E1 24.9554,E2 344.0509} C_DIS
LIN {X -32.6954,Y 103.2325,Z 114,A 103.2497,B 24.9269,C -1.9743,E1 24.9509,E2 342.3821} C_DIS
LIN {X -35.2038,Y 102.4042,Z 114,A 104.6727,B 24.9269,C -1.9735,E1 24.9472,E2 340.9581} C_DIS
LIN {X -37.7278,Y 101.5015,Z 114,A 106.2318,B 24.9267,C -1.9772,E1 24.943,E2 339.3871} C_DIS
LIN {X -40.8343,Y 100.2899,Z 114,A 107.8303,B 24.9274,C -1.9683,E1 24.9389,E2 337.8062} C_DIS
LIN {X -43.2746,Y 99.2614,Z 114,A 109.2519,B 24.9274,C -1.9671,E1 24.9353,E2 336.3842} C_DIS
LIN {X -45.6896,Y 98.1732,Z 114,A 110.7038,B 24.9274,C -1.9669,E1 24.9316,E2 334.9293} C_DIS
LIN {X -48.7016,Y 96.7165,Z 114,A 112.43,B 24.9278,C -1.9623,E1 24.9273,E2 333.2094} C_DIS
LIN {X -51.055,Y 95.4952,Z 114,A 113.8382,B 24.928,C -1.9602,E1 24.9238,E2 331.8024} C_DIS
LIN {X -53.3782,Y 94.2163,Z 114,A 115.2469,B 24.9281,C -1.9579,E1 24.9204,E2 330.3951} C_DIS
LIN {X -55.6695,Y 92.8809,Z 114,A 116.657,B 24.9283,C -1.9556,E1 24.917,E2 328.9861} C_DIS
LIN {X -57.9273,Y 91.4897,Z 114,A 118.0659,B 24.9285,C -1.9532,E1 24.9137,E2 327.5785} C_DIS
LIN {X -60.1502,Y 90.0438,Z 114,A 119.4751,B 24.9287,C -1.9507,E1 24.9104,E2 326.1706} C_DIS
LIN {X -62.3607,Y 88.5273,Z 114,A 120.8971,B 24.9289,C -1.948,E1 24.9071,E2 324.7502} C_DIS
LIN {X -64.5063,Y 86.9764,Z 114,A 122.4375,B 24.9287,C -1.9504,E1 24.9036,E2 323.1986} C_DIS
LIN {X -67.1346,Y 84.9615,Z 114,A 124.1296,B 24.9291,C -1.9444,E1 24.8999,E2 321.5146} C_DIS
LIN {X -69.9601,Y 82.6512,Z 114,A 126.1023,B 24.9293,C -1.9417,E1 24.8957,E2 319.5408} C_DIS
LIN {X -72.4871,Y 80.4441,Z 114,A 127.9527,B 24.9294,C -1.9405,E1 24.8918,E2 317.686} C_DIS
LIN {X -75.1378,Y 77.9732,Z 114,A 129.785,B 24.93,C -1.9327,E1 24.8881,E2 315.8647} C_DIS
LIN {X -77.7004,Y 75.4209,Z 114,A 131.746,B 24.9302,C -1.9298,E1 24.8843,E2 313.9023} C_DIS
LIN {X -79.9743,Y 73.0047,Z 114,A 133.5756,B 24.9302,C -1.9282,E1 24.8808,E2 312.0683} C_DIS
LIN {X -82.4224,Y 70.2287,Z 114,A 135.4437,B 24.9309,C -1.9197,E1 24.8774,E2 310.212} C_DIS
LIN {X -84.7256,Y 67.433,Z 114,A 137.4076,B 24.9311,C -1.9165,E1 24.8739,E2 308.2467} C_DIS
LIN {X -86.5325,Y 65.0971,Z 114,A 138.8925,B 24.9317,C -1.9093,E1 24.8714,E2 306.7718} C_DIS
LIN {X -88.1621,Y 62.8725,Z 114,A 140.3332,B 24.932,C -1.9046,E1 24.8691,E2 305.3352} C_DIS
LIN {X -89.648,Y 60.7351,Z 114,A 141.7417,B 24.9322,C -1.902,E1 24.8669,E2 303.9262} C_DIS
LIN {X -91.1069,Y 58.5239,Z 114,A 143.152,B 24.9324,C -1.8983,E1 24.8647,E2 302.5174} C_DIS
LIN {X -92.5108,Y 56.2785,Z 114,A 144.6201,B 24.9326,C -1.8968,E1 24.8626,E2 301.0454} C_DIS
LIN {X -94.2195,Y 53.3726,Z 114,A 146.3457,B 24.9331,C -1.8894,E1 24.8602,E2 299.3285} C_DIS
LIN {X -95.4986,Y 51.0487,Z 114,A 147.7592,B 24.9333,C -1.8857,E1 24.8583,E2 297.9164} C_DIS
LIN {X -96.7202,Y 48.6943,Z 114,A 149.1718,B 24.9336,C -1.8818,E1 24.8565,E2 296.5054} C_DIS
LIN {X -98.105,Y 45.8361,Z 114,A 150.8993,B 24.9338,C -1.8786,E1 24.8544,E2 294.7763} C_DIS
LIN {X -99.466,Y 42.8053,Z 114,A 152.7103,B 24.9341,C -1.8752,E1 24.8524,E2 292.9634} C_DIS
LIN {X -100.4652,Y 40.4036,Z 114,A 154.0365,B 24.9345,C -1.8691,E1 24.851,E2 291.6444} C_DIS
LIN {X -101.5029,Y 37.724,Z 114,A 155.548,B 24.9349,C -1.864,E1 24.8495,E2 290.1365} C_DIS
LIN {X -102.3964,Y 35.2269,Z 114,A 156.9624,B 24.9351,C -1.86,E1 24.8482,E2 288.7235} C_DIS
LIN {X -103.2283,Y 32.7086,Z 114,A 158.4103,B 24.9353,C -1.8573,E1 24.847,E2 287.2739} C_DIS
LIN {X -104.0022,Y 30.1579,Z 114,A 159.7943,B 24.9357,C -1.8518,E1 24.8459,E2 285.8948} C_DIS
LIN {X -104.7146,Y 27.5824,Z 114,A 161.2166,B 24.936,C -1.8477,E1 24.8448,E2 284.4743} C_DIS
LIN {X -105.3576,Y 25.0142,Z 114,A 162.8069,B 24.9358,C -1.8503,E1 24.8438,E2 282.8685} C_DIS
LIN {X -106.0756,Y 21.7597,Z 114,A 164.3928,B 24.9367,C -1.838,E1 24.8429,E2 281.3025} C_DIS
LIN {X -106.5676,Y 19.2057,Z 114,A 165.7899,B 24.9369,C -1.8343,E1 24.8422,E2 279.9058} C_DIS
LIN {X -107.0051,Y 16.5961,Z 114,A 167.2114,B 24.9372,C -1.8306,E1 24.8415,E2 278.4848} C_DIS
LIN {X -107.3846,Y 13.9305,Z 114,A 168.6211,B 24.9375,C -1.8255,E1 24.841,E2 277.0789} C_DIS
LIN {X -107.7673,Y 10.5887,Z 114,A 170.729,B 24.9371,C -1.8319,E1 24.8404,E2 274.943} C_DIS
LIN {X -108.0825,Y 6.6418,Z 114,A 172.753,B 24.9377,C -1.8224,E1 24.84,E2 272.9294} C_DIS
LIN {X -108.255,Y 2.5954,Z 114,A 174.679,B 24.9388,C -1.8074,E1 24.8398,E2 271.0277} C_DIS
LIN {X -108.2849,Y -0.2562,Z 114,A 176.3329,B 24.9388,C -1.8079,E1 24.8398,E2 269.3625} C_DIS
LIN {X -108.2168,Y -3.8629,Z 114,A 178.2842,B 24.939,C -1.8033,E1 24.8399,E2 267.4105} C_DIS
LIN {X -108.0206,Y -7.5577,Z 114,A -179.8082,B 24.9396,C -1.7952,E1 24.8403,E2 265.5109} C_DIS
LIN {X -107.7013,Y -11.222,Z 114,A -177.8262,B 24.9399,C -1.7903,E1 24.8408,E2 263.5286} C_DIS
LIN {X -107.2727,Y -14.7744,Z 114,A -176.1223,B 24.9408,C -1.7771,E1 24.8414,E2 261.8459} C_DIS
LIN {X -106.9045,Y -17.2429,Z 114,A -174.7003,B 24.9408,C -1.7767,E1 24.842,E2 260.4163} C_DIS
LIN {X -106.454,Y -19.836,Z 114,A -173.1564,B 24.9408,C -1.778,E1 24.8428,E2 258.8602} C_DIS
LIN {X -105.8048,Y -23.0403,Z 114,A -171.5531,B 24.9414,C -1.7679,E1 24.8437,E2 257.2717} C_DIS
LIN {X -105.2028,Y -25.6493,Z 114,A -170.0376,B 24.9414,C -1.7672,E1 24.8447,E2 255.7489} C_DIS
LIN {X -104.3653,Y -28.8762,Z 114,A -168.2966,B 24.9419,C -1.7609,E1 24.8459,E2 254.0129} C_DIS
LIN {X -103.6228,Y -31.4367,Z 114,A -166.9289,B 24.9423,C -1.755,E1 24.847,E2 252.6514} C_DIS
LIN {X -102.8217,Y -33.9652,Z 114,A -165.5151,B 24.9425,C -1.7511,E1 24.8482,E2 251.2386} C_DIS
LIN {X -101.7598,Y -37.0197,Z 114,A -163.7475,B 24.9427,C -1.7482,E1 24.8499,E2 249.468} C_DIS
LIN {X -100.5432,Y -40.2121,Z 114,A -161.9748,B 24.9432,C -1.7415,E1 24.8517,E2 247.7013} C_DIS
LIN {X -99.5281,Y -42.6628,Z 114,A -160.5611,B 24.9434,C -1.7379,E1 24.8532,E2 246.2885} C_DIS
LIN {X -98.441,Y -45.1142,Z 114,A -159.1385,B 24.9437,C -1.7339,E1 24.8548,E2 244.8674} C_DIS
LIN {X -97.1247,Y -47.8787,Z 114,A -157.446,B 24.9437,C -1.7321,E1 24.8569,E2 243.1701} C_DIS
LIN {X -95.811,Y -50.4555,Z 114,A -155.9785,B 24.9442,C -1.7255,E1 24.8588,E2 241.7105} C_DIS
LIN {X -94.5569,Y -52.7685,Z 114,A -154.4946,B 24.9442,C -1.7252,E1 24.8608,E2 240.2195} C_DIS
LIN {X -92.8784,Y -55.6736,Z 114,A -152.7786,B 24.9447,C -1.7181,E1 24.8632,E2 238.5114} C_DIS
LIN {X -91.4869,Y -57.9319,Z 114,A -151.1997,B 24.9445,C -1.7211,E1 24.8656,E2 236.9173} C_DIS
LIN {X -89.6458,Y -60.7382,Z 114,A -149.5204,B 24.945,C -1.7129,E1 24.8682,E2 235.2494} C_DIS
LIN {X -87.7651,Y -63.4289,Z 114,A -147.8333,B 24.9454,C -1.7066,E1 24.8709,E2 233.5689} C_DIS
LIN {X -85.9803,Y -65.8256,Z 114,A -146.401,B 24.946,C -1.697,E1 24.8733,E2 232.1526} C_DIS
LIN {X -84.3481,Y -67.9046,Z 114,A -144.7324,B 24.9456,C -1.704,E1 24.8762,E2 230.4595} C_DIS
LIN {X -82.1964,Y -70.4939,Z 114,A -142.8838,B 24.9456,C -1.7025,E1 24.8795,E2 228.6061} C_DIS
LIN {X -79.7832,Y -73.2131,Z 114,A -141.0523,B 24.9462,C -1.6946,E1 24.883,E2 226.7852} C_DIS
LIN {X -77.2799,Y -75.8515,Z 114,A -139.0805,B 24.9463,C -1.6922,E1 24.8868,E2 224.8106} C_DIS
LIN {X -74.9041,Y -78.1985,Z 114,A -137.2525,B 24.9464,C -1.6909,E1 24.8905,E2 222.9781} C_DIS
LIN {X -72.2268,Y -80.6771,Z 114,A -135.3985,B 24.9469,C -1.684,E1 24.8943,E2 221.133} C_DIS
LIN {X -69.4714,Y -83.0624,Z 114,A -133.4247,B 24.9469,C -1.6821,E1 24.8985,E2 219.1562} C_DIS
LIN {X -66.8643,Y -85.1752,Z 114,A -131.7188,B 24.9474,C -1.6761,E1 24.9022,E2 217.4582} C_DIS
LIN {X -64.2227,Y -87.184,Z 114,A -129.8957,B 24.9474,C -1.6756,E1 24.9063,E2 215.6297} C_DIS
LIN {X -61.8612,Y -88.8747,Z 114,A -128.4457,B 24.9478,C -1.6696,E1 24.9095,E2 214.189} C_DIS
LIN {X -59.2942,Y -90.6082,Z 114,A -126.7719,B 24.9478,C -1.6684,E1 24.9134,E2 212.5126} C_DIS
LIN {X -56.5056,Y -92.3727,Z 114,A -124.9611,B 24.9478,C -1.6683,E1 24.9178,E2 210.6964} C_DIS
LIN {X -53.9761,Y -93.8728,Z 114,A -123.4855,B 24.9482,C -1.6628,E1 24.9213,E2 209.2292} C_DIS
LIN {X -51.3364,Y -95.3425,Z 114,A -121.844,B 24.9482,C -1.6624,E1 24.9253,E2 207.5842} C_DIS
LIN {X -48.6795,Y -96.7277,Z 114,A -120.2922,B 24.9484,C -1.659,E1 24.9292,E2 206.0362} C_DIS
LIN {X -46.2957,Y -97.8911,Z 114,A -118.885,B 24.9485,C -1.6574,E1 24.9327,E2 204.6291} C_DIS
LIN {X -43.3612,Y -99.2236,Z 114,A -117.1453,B 24.9485,C -1.657,E1 24.9372,E2 202.8864} C_DIS
LIN {X -40.8527,Y -100.2824,Z 114,A -115.7198,B 24.9487,C -1.6549,E1 24.9408,E2 201.4626} C_DIS
LIN {X -37.9489,Y -101.4178,Z 114,A -114.0594,B 24.9487,C -1.6537,E1 24.9452,E2 199.8014} C_DIS
LIN {X -34.7009,Y -102.5737,Z 114,A -112.2182,B 24.9488,C -1.6529,E1 24.95,E2 197.9587} C_DIS
LIN {X -32.1055,Y -103.4154,Z 114,A -110.786,B 24.9489,C -1.6513,E1 24.9538,E2 196.5276} C_DIS
LIN {X -29.4361,Y -104.2067,Z 114,A -109.2527,B 24.9489,C -1.6527,E1 24.958,E2 194.9885} C_DIS
LIN {X -25.9181,Y -105.1372,Z 114,A -107.3217,B 24.9489,C -1.6518,E1 24.9632,E2 193.0568} C_DIS
LIN {X -23.0465,Y -105.8035,Z 114,A -105.8394,B 24.9491,C -1.6479,E1 24.9672,E2 191.5818} C_DIS
LIN {X -20.4935,Y -106.3274,Z 114,A -104.4591,B 24.9491,C -1.6474,E1 24.971,E2 190.2012} C_DIS
LIN {X -17.8829,Y -106.7975,Z 114,A -103.0546,B 24.9491,C -1.647,E1 24.9748,E2 188.7963} C_DIS
LIN {X -15.2133,Y -107.2104,Z 114,A -101.6245,B 24.9491,C -1.6467,E1 24.9788,E2 187.3657} C_DIS
LIN {X -12.6289,Y -107.5454,Z 114,A -100.2298,B 24.9491,C -1.6471,E1 24.9827,E2 185.9691} C_DIS
LIN {X -9.9746,Y -107.824,Z 114,A -98.8212,B 24.9491,C -1.6468,E1 24.9866,E2 184.5604} C_DIS
LIN {X -7.3305,Y -108.036,Z 114,A -97.4177,B 24.9491,C -1.6468,E1 24.9905,E2 183.1564} C_DIS
LIN {X -4.6358,Y -108.1851,Z 114,A -96.0012,B 24.9492,C -1.6465,E1 24.9944,E2 181.7403} C_DIS
LIN {X -2.0197,Y -108.2656,Z 114,A -94.6166,B 24.9492,C -1.6467,E1 24.9983,E2 180.3552} C_DIS
LIN {X 0.7824,Y -108.2811,Z 114,A -93.1783,B 24.9492,C -1.6452,E1 25.0023,E2 178.9204} C_DIS
Enddeposition()
LIN {X 0.8034,Y -114.4827,Z 115,A -93.2941,B 24.9556,C -1.5397,E1 25.0013,E2 179.2861} C_DIS
Startdeposition()
$VEL.CP = VEL_PRINT
LIN {X -2.5968,Y -114.457,Z 115,A -95.2692,B 24.9563,C -1.5274,E1 24.9957,E2 181.2905} C_DIS
LIN {X -5.4049,Y -114.3588,Z 115,A -96.6861,B 24.9563,C -1.5268,E1 24.9917,E2 182.7091} C_DIS
LIN {X -8.2098,Y -114.1917,Z 115,A -98.0807,B 24.9563,C -1.5273,E1 24.9879,E2 184.103} C_DIS
LIN {X -10.6336,Y -113.9906,Z 115,A -99.354,B 24.9564,C -1.525,E1 24.9843,E2 185.3824} C_DIS
LIN {X -13.803,Y -113.6514,Z 115,A -100.8929,B 24.9563,C -1.5276,E1 24.98,E2 186.9161} C_DIS
LIN {X -16.7988,Y -113.2484,Z 115,A -102.4065,B 24.9563,C -1.5279,E1 24.9759,E2 188.4302} C_DIS
LIN {X -19.573,Y -112.8021,Z 115,A -103.8134,B 24.9563,C -1.5283,E1 24.972,E2 189.8375} C_DIS
LIN {X -22.1263,Y -112.328,Z 115,A -105.1269,B 24.9563,C -1.5283,E1 24.9684,E2 191.1527} C_DIS
LIN {X -25.0844,Y -111.7058,Z 115,A -106.6286,B 24.9562,C -1.5294,E1 24.9643,E2 192.6535} C_DIS
LIN {X -27.8182,Y -111.0565,Z 115,A -108.0364,B 24.9562,C -1.5301,E1 24.9605,E2 194.0616} C_DIS
LIN {X -30.3297,Y -110.3959,Z 115,A -109.338,B 24.9561,C -1.5308,E1 24.957,E2 195.3634} C_DIS
LIN {X -33.0299,Y -109.6183,Z 115,A -110.7461,B 24.9561,C -1.5317,E1 24.9532,E2 196.7717} C_DIS
LIN {X -35.9127,Y -108.7092,Z 115,A -112.2618,B 24.956,C -1.5327,E1 24.9491,E2 198.2877} C_DIS
LIN {X -38.5697,Y -107.7951,Z 115,A -113.6703,B 24.956,C -1.5338,E1 24.9454,E2 199.6963} C_DIS
LIN {X -41.0044,Y -106.8915,Z 115,A -114.9728,B 24.9559,C -1.535,E1 24.942,E2 200.9988} C_DIS
LIN {X -43.8125,Y -105.7727,Z 115,A -116.4889,B 24.9558,C -1.5363,E1 24.9381,E2 202.515} C_DIS
LIN {X -46.3951,Y -104.6657,Z 115,A -117.8984,B 24.9557,C -1.5377,E1 24.9345,E2 203.9246} C_DIS
LIN {X -48.9497,Y -103.4955,Z 115,A -119.3082,B 24.9557,C -1.5392,E1 24.9309,E2 205.3344} C_DIS
LIN {X -51.2841,Y -102.3577,Z 115,A -120.6112,B 24.9555,C -1.5407,E1 24.9277,E2 206.6373} C_DIS
LIN {X -53.7807,Y -101.0683,Z 115,A -122.0342,B 24.9555,C -1.5418,E1 24.9241,E2 208.0615} C_DIS
LIN {X -56.2448,Y -99.718,Z 115,A -123.432,B 24.9553,C -1.5441,E1 24.9207,E2 209.4579} C_DIS
LIN {X -58.8584,Y -98.1993,Z 115,A -124.9494,B 24.9553,C -1.5461,E1 24.9171,E2 210.9751} C_DIS
LIN {X -61.07,Y -96.8381,Z 115,A -126.264,B 24.9551,C -1.5475,E1 24.914,E2 212.2906} C_DIS
LIN {X -63.1584,Y -95.488,Z 115,A -127.5481,B 24.9551,C -1.5478,E1 24.911,E2 213.5781} C_DIS
LIN {X -65.9229,Y -93.6033,Z 115,A -129.1828,B 24.9549,C -1.5522,E1 24.9072,E2 215.2079} C_DIS
LIN {X -68.0284,Y -92.0831,Z 115,A -130.4998,B 24.9548,C -1.5538,E1 24.9042,E2 216.5259} C_DIS
LIN {X -70.0425,Y -90.5594,Z 115,A -131.7944,B 24.9548,C -1.5548,E1 24.9014,E2 217.8227} C_DIS
LIN {X -72.4647,Y -88.6342,Z 115,A -133.311,B 24.9545,C -1.559,E1 24.8981,E2 219.335} C_DIS
LIN {X -74.7802,Y -86.691,Z 115,A -134.8299,B 24.9543,C -1.5616,E1 24.8949,E2 220.8536} C_DIS
LIN {X -77.7635,Y -84.0238,Z 115,A -136.8542,B 24.9541,C -1.5648,E1 24.8907,E2 222.8784} C_DIS
LIN {X -79.8021,Y -82.0901,Z 115,A -138.2669,B 24.954,C -1.5674,E1 24.8878,E2 224.2907} C_DIS
LIN {X -81.7926,Y -80.1069,Z 115,A -139.6795,B 24.9538,C -1.5702,E1 24.885,E2 225.7027} C_DIS
LIN {X -83.7339,Y -78.0755,Z 115,A -141.0925,B 24.9536,C -1.573,E1 24.8823,E2 227.1151} C_DIS
LIN {X -85.7668,Y -75.8384,Z 115,A -142.6001,B 24.9534,C -1.5766,E1 24.8795,E2 228.6208} C_DIS
LIN {X -87.4641,Y -73.8728,Z 115,A -143.919,B 24.9533,C -1.5789,E1 24.8771,E2 229.9404} C_DIS
LIN {X -89.3847,Y -71.5387,Z 115,A -145.4268,B 24.9531,C -1.5827,E1 24.8745,E2 231.4462} C_DIS
LIN {X -91.8294,Y -68.3704,Z 115,A -147.4531,B 24.9528,C -1.5867,E1 24.871,E2 233.4727} C_DIS
LIN {X -93.4796,Y -66.0962,Z 115,A -148.8541,B 24.9526,C -1.5904,E1 24.8688,E2 234.8716} C_DIS
LIN {X -95.1929,Y -63.6059,Z 115,A -150.3752,B 24.9524,C -1.5939,E1 24.8664,E2 236.3919} C_DIS
LIN {X -96.6102,Y -61.4298,Z 115,A -151.6952,B 24.9522,C -1.5965,E1 24.8644,E2 237.7123} C_DIS
LIN {X -98.1993,Y -58.8584,Z 115,A -153.2038,B 24.952,C -1.6007,E1 24.8622,E2 239.2188} C_DIS
LIN {X -99.6142,Y -56.4307,Z 115,A -154.6181,B 24.9518,C -1.6042,E1 24.8602,E2 240.6322} C_DIS
LIN {X -100.8675,Y -54.1562,Z 115,A -155.9384,B 24.9516,C -1.6069,E1 24.8585,E2 241.9529} C_DIS
LIN {X -102.0758,Y -51.8413,Z 115,A -157.2832,B 24.9515,C -1.609,E1 24.8567,E2 243.2998} C_DIS
LIN {X -103.4955,Y -48.9497,Z 115,A -158.8625,B 24.9511,C -1.6149,E1 24.8548,E2 244.8738} C_DIS
LIN {X -104.5782,Y -46.5892,Z 115,A -160.1704,B 24.9509,C -1.6183,E1 24.8533,E2 246.1806} C_DIS
LIN {X -105.7727,Y -43.8125,Z 115,A -161.6927,B 24.9507,C -1.6223,E1 24.8517,E2 247.7019} C_DIS
LIN {X -106.8161,Y -41.2035,Z 115,A -163.1076,B 24.9505,C -1.6261,E1 24.8502,E2 249.1156} C_DIS
LIN {X -107.7221,Y -38.7697,Z 115,A -164.416,B 24.9502,C -1.6296,E1 24.849,E2 250.423} C_DIS
LIN {X -108.6412,Y -36.1144,Z 115,A -165.7896,B 24.9499,C -1.6351,E1 24.8478,E2 251.7913} C_DIS
LIN {X -109.3888,Y -33.779,Z 115,A -167.142,B 24.9499,C -1.6339,E1 24.8466,E2 253.1544} C_DIS
LIN {X -110.3404,Y -30.5353,Z 115,A -168.7696,B 24.9495,C -1.6416,E1 24.8454,E2 254.7731} C_DIS
LIN {X -111.0565,Y -27.8182,Z 115,A -170.1853,B 24.9493,C -1.6456,E1 24.8444,E2 256.1876} C_DIS
LIN {X -111.6579,Y -25.2918,Z 115,A -171.4939,B 24.949,C -1.6493,E1 24.8436,E2 257.495} C_DIS
LIN {X -112.2449,Y -22.544,Z 115,A -172.9222,B 24.9488,C -1.6528,E1 24.8427,E2 258.9233} C_DIS
LIN {X -112.9986,Y -18.3973,Z 115,A -175.0461,B 24.9484,C -1.6589,E1 24.8417,E2 261.0453} C_DIS
LIN {X -113.4161,Y -15.6186,Z 115,A -176.4621,B 24.9482,C -1.663,E1 24.8412,E2 262.46} C_DIS
LIN {X -113.79,Y -12.6191,Z 115,A -177.9726,B 24.9479,C -1.6679,E1 24.8407,E2 263.9679} C_DIS
LIN {X -114.0459,Y -10.0348,Z 115,A -179.2699,B 24.9476,C -1.6722,E1 24.8403,E2 265.2627} C_DIS
LIN {X -114.2721,Y -7.0205,Z 115,A 179.1951,B 24.9474,C -1.6762,E1 24.84,E2 266.7975} C_DIS
LIN {X -114.41,Y -4.214,Z 115,A 177.779,B 24.9471,C -1.6803,E1 24.8399,E2 268.2122} C_DIS
LIN {X -114.479,Y -1.4049,Z 115,A 176.3389,B 24.9469,C -1.6835,E1 24.8398,E2 269.6532} C_DIS
LIN {X -114.4817,Y 1.0162,Z 115,A 175.1108,B 24.9467,C -1.6868,E1 24.8398,E2 270.8809} C_DIS
LIN {X -114.4257,Y 3.7039,Z 115,A 173.7886,B 24.9463,C -1.6921,E1 24.8399,E2 272.1984} C_DIS
LIN {X -114.3057,Y 6.4136,Z 115,A 172.3597,B 24.9463,C -1.6937,E1 24.8401,E2 273.6321} C_DIS
LIN {X -114.0654,Y 9.8227,Z 115,A 170.6985,B 24.9458,C -1.7012,E1 24.8405,E2 275.2855} C_DIS
LIN {X -113.8122,Y 12.4073,Z 115,A 169.3895,B 24.9455,C -1.7051,E1 24.8408,E2 276.5931} C_DIS
LIN {X -113.5251,Y 14.7974,Z 115,A 168.1135,B 24.9455,C -1.7062,E1 24.8413,E2 277.8741} C_DIS
LIN {X -113.0338,Y 18.1873,Z 115,A 166.4501,B 24.945,C -1.7137,E1 24.842,E2 279.5295} C_DIS
LIN {X -112.5534,Y 20.9558,Z 115,A 165.034,B 24.9447,C -1.7179,E1 24.8427,E2 280.9441} C_DIS
LIN {X -112.048,Y 23.5031,Z 115,A 163.725,B 24.9444,C -1.7217,E1 24.8434,E2 282.2516} C_DIS
LIN {X -111.5205,Y 25.8865,Z 115,A 162.4396,B 24.9444,C -1.7231,E1 24.8442,E2 283.5412} C_DIS
LIN {X -110.7598,Y 28.9727,Z 115,A 160.8932,B 24.9439,C -1.7299,E1 24.8453,E2 285.0803} C_DIS
LIN {X -110.0154,Y 31.6822,Z 115,A 159.4771,B 24.9436,C -1.734,E1 24.8463,E2 286.4949} C_DIS
LIN {X -109.1417,Y 34.5759,Z 115,A 157.954,B 24.9434,C -1.7384,E1 24.8476,E2 288.0164} C_DIS
LIN {X -108.2603,Y 37.244,Z 115,A 156.538,B 24.9431,C -1.7424,E1 24.8488,E2 289.4308} C_DIS
LIN {X -107.3866,Y 39.6896,Z 115,A 155.2297,B 24.9429,C -1.7461,E1 24.8501,E2 290.7377} C_DIS
LIN {X -106.3803,Y 42.313,Z 115,A 153.8139,B 24.9426,C -1.7501,E1 24.8515,E2 292.1519} C_DIS
LIN {X -105.3098,Y 44.911,Z 115,A 152.3856,B 24.9424,C -1.7536,E1 24.8531,E2 293.5799} C_DIS
LIN {X -104.0884,Y 47.676,Z 115,A 150.8757,B 24.9421,C -1.7583,E1 24.8548,E2 295.0869} C_DIS
LIN {X -102.9793,Y 50.0242,Z 115,A 149.5547,B 24.9419,C -1.7614,E1 24.8564,E2 296.4078} C_DIS
LIN {X -101.6237,Y 52.726,Z 115,A 148.0449,B 24.9415,C -1.766,E1 24.8583,E2 297.9146} C_DIS
LIN {X -100.4007,Y 55.0169,Z 115,A 146.757,B 24.9413,C -1.7703,E1 24.86,E2 299.1991} C_DIS
LIN {X -99.0203,Y 57.4643,Z 115,A 145.3089,B 24.9411,C -1.7727,E1 24.862,E2 300.6489} C_DIS
LIN {X -97.4696,Y 60.059,Z 115,A 143.7994,B 24.9408,C -1.7772,E1 24.8642,E2 302.1555} C_DIS
LIN {X -95.9663,Y 62.4329,Z 115,A 142.3845,B 24.9406,C -1.7808,E1 24.8663,E2 303.5689} C_DIS
LIN {X -94.4052,Y 64.7693,Z 115,A 140.9698,B 24.9403,C -1.7844,E1 24.8685,E2 304.982} C_DIS
LIN {X -92.911,Y 66.8932,Z 115,A 139.6621,B 24.9401,C -1.7877,E1 24.8706,E2 306.2883} C_DIS
LIN {X -91.1134,Y 69.3235,Z 115,A 138.1406,B 24.9398,C -1.7915,E1 24.8732,E2 307.8082} C_DIS
LIN {X -89.5167,Y 71.3716,Z 115,A 136.8208,B 24.9397,C -1.7942,E1 24.8755,E2 309.1277} C_DIS
LIN {X -87.781,Y 73.4956,Z 115,A 135.4468,B 24.9394,C -1.7977,E1 24.8779,E2 310.4996} C_DIS
LIN {X -85.9069,Y 75.678,Z 115,A 133.9923,B 24.9392,C -1.8008,E1 24.8806,E2 311.9533} C_DIS
LIN {X -83.8798,Y 77.9204,Z 115,A 132.4841,B 24.9389,C -1.8048,E1 24.8834,E2 313.4586} C_DIS
LIN {X -81.9423,Y 79.9554,Z 115,A 131.07,B 24.9387,C -1.808,E1 24.8862,E2 314.8713} C_DIS
LIN {X -80.1303,Y 81.7695,Z 115,A 129.7637,B 24.9386,C -1.8102,E1 24.8887,E2 316.1779} C_DIS
LIN {X -78.0755,Y 83.7339,Z 115,A 128.3373,B 24.9384,C -1.8134,E1 24.8916,E2 317.6025} C_DIS
LIN {X -75.8384,Y 85.7668,Z 115,A 126.8298,B 24.9381,C -1.8171,E1 24.8948,E2 319.1072} C_DIS
LIN {X -73.8728,Y 87.4641,Z 115,A 125.5108,B 24.938,C -1.8193,E1 24.8976,E2 320.4261} C_DIS
LIN {X -71.5387,Y 89.3847,Z 115,A 124.0037,B 24.9377,C -1.8228,E1 24.9008,E2 321.9305} C_DIS
LIN {X -69.3235,Y 91.1134,Z 115,A 122.5911,B 24.9375,C -1.8256,E1 24.9039,E2 323.3417} C_DIS
LIN {X -67.0666,Y 92.7873,Z 115,A 121.1784,B 24.9373,C -1.8282,E1 24.9071,E2 324.7531} C_DIS
LIN {X -64.9441,Y 94.2837,Z 115,A 119.873,B 24.9372,C -1.8306,E1 24.9101,E2 326.0572} C_DIS
LIN {X -62.4329,Y 95.9663,Z 115,A 118.3538,B 24.937,C -1.8333,E1 24.9137,E2 327.575} C_DIS
LIN {X -60.059,Y 97.4696,Z 115,A 116.9419,B 24.9368,C -1.8357,E1 24.917,E2 328.9856} C_DIS
LIN {X -58.0874,Y 98.655,Z 115,A 115.724,B 24.9368,C -1.8352,E1 24.9199,E2 330.2085} C_DIS
LIN {X -55.2041,Y 100.2991,Z 115,A 114.1184,B 24.9365,C -1.8403,E1 24.9238,E2 331.8065} C_DIS
LIN {X -52.9144,Y 101.5245,Z 115,A 112.8142,B 24.9364,C -1.8423,E1 24.927,E2 333.1095} C_DIS
LIN {X -50.4069,Y 102.7925,Z 115,A 111.3902,B 24.9363,C -1.8439,E1 24.9306,E2 334.5337} C_DIS
LIN {X -47.8691,Y 103.9986,Z 115,A 109.9919,B 24.9361,C -1.8464,E1 24.9341,E2 335.9295} C_DIS
LIN {X -45.3024,Y 105.142,Z 115,A 108.5685,B 24.936,C -1.8478,E1 24.9378,E2 337.353} C_DIS
LIN {X -42.7084,Y 106.2221,Z 115,A 107.1578,B 24.9359,C -1.8496,E1 24.9414,E2 338.7626} C_DIS
LIN {X -39.8896,Y 107.3137,Z 115,A 105.6534,B 24.9357,C -1.8519,E1 24.9453,E2 340.2646} C_DIS
LIN {X -37.4449,Y 108.1898,Z 115,A 104.3377,B 24.9357,C -1.8529,E1 24.9488,E2 341.5805} C_DIS
LIN {X -34.5759,Y 109.1417,Z 115,A 102.8334,B 24.9355,C -1.855,E1 24.9528,E2 343.0825} C_DIS
LIN {X -31.887,Y 109.9574,Z 115,A 101.424,B 24.9354,C -1.8565,E1 24.9566,E2 344.4909} C_DIS
LIN {X -29.179,Y 110.7068,Z 115,A 100.0145,B 24.9354,C -1.8578,E1 24.9604,E2 345.8993} C_DIS
LIN {X -26.6601,Y 111.3391,Z 115,A 98.7122,B 24.9352,C -1.859,E1 24.9639,E2 347.2007} C_DIS
LIN {X -23.9197,Y 111.9598,Z 115,A 97.3032,B 24.9352,C -1.8601,E1 24.9677,E2 348.6087} C_DIS
LIN {X -20.9558,Y 112.5534,Z 115,A 95.7877,B 24.9351,C -1.8612,E1 24.9719,E2 350.1234} C_DIS
LIN {X -18.3973,Y 112.9986,Z 115,A 94.4733,B 24.9351,C -1.8615,E1 24.9755,E2 351.4381} C_DIS
LIN {X -15.6186,Y 113.4161,Z 115,A 93.0651,B 24.935,C -1.8624,E1 24.9794,E2 352.8455} C_DIS
LIN {X -12.6191,Y 113.79,Z 115,A 91.563,B 24.9349,C -1.8637,E1 24.9835,E2 354.3455} C_DIS
LIN {X -8.6345,Y 114.1604,Z 115,A 89.5458,B 24.9349,C -1.864,E1 24.9892,E2 356.3629} C_DIS
LIN {X -6.0075,Y 114.3281,Z 115,A 88.2011,B 24.9349,C -1.8634,E1 24.9929,E2 357.7094} C_DIS
LIN {X -3.0225,Y 114.4466,Z 115,A 86.7312,B 24.9349,C -1.8649,E1 24.997,E2 359.1761} C_DIS
LIN {X -0.2129,Y 114.4863,Z 115,A 85.3241,B 24.9348,C -1.8652,E1 25.0009,E2 360.5825} C_DIS
Enddeposition()
END
